// Clear works correctly after popping elements
METHOD ClearAfterPop
VAR
	ReturnedElement : DINT;
END_VAR
IF TestSuite.Test(__POUNAME()).ExecuteTest() THEN
	// Arrange - Push and then pop elements
	fbAnyBuffer.Clear();
	testElement := DINT#100;
	fbAnyBuffer.PushLeft(element := testElement);
	testElement := DINT#200;
	fbAnyBuffer.PushLeft(element := testElement);
	testElement := DINT#200;
	fbAnyBuffer.PushLeft(element := testElement);
	fbAnyBuffer.PopLeft(element := ReturnedElement);
	fbAnyBuffer.PopLeft(element := ReturnedElement);

	// Act
	Success := fbAnyBuffer.Clear();

	// Assert
	TestSuite.Test(__POUNAME()).AssertEqual(TEST_BOOL_TRUE, Success);
	TEST_DINT := 0;
	TestSuite.Test(__POUNAME()).AssertEqual(TEST_DINT, fbAnyBuffer.Metadata.elementCount);
	TestSuite.Test(__POUNAME()).AssertEqual(TEST_DINT, RawBuffer[TEST_LL+0]);
END_IF
END_METHOD

// Clear works correctly after pushing elements
METHOD ClearAfterPush
IF TestSuite.Test(__POUNAME()).ExecuteTest() THEN
	// Arrange - Push some elements first
	fbAnyBuffer.Clear();
	testElement := DINT#100;
	fbAnyBuffer.PushLeft(element := testElement);
	fbAnyBuffer.PushLeft(element := testElement);
	fbAnyBuffer.PushLeft(element := testElement);

	// Act
	Success := fbAnyBuffer.Clear();

	// Assert
	TestSuite.Test(__POUNAME()).AssertEqual(TEST_BOOL_TRUE, Success);
	TEST_DINT := 0;
	TestSuite.Test(__POUNAME()).AssertEqual(TEST_DINT, fbAnyBuffer.Metadata.elementCount);
	TestSuite.Test(__POUNAME()).AssertEqual(TEST_DINT, RawBuffer[TEST_LL+0]);
	TestSuite.Test(__POUNAME()).AssertEqual(TEST_DINT, RawBuffer[TEST_LL+1]);
	TestSuite.Test(__POUNAME()).AssertEqual(TEST_DINT, RawBuffer[TEST_LL+2]);
END_IF
END_METHOD

// Clear on already-empty buffer returns TRUE
METHOD ClearEmptyBuffer
IF TestSuite.Test(__POUNAME()).ExecuteTest() THEN
	// Arrange - Buffer is already empty (elementCount = 0)
	fbAnyBuffer.Clear();

	// Act - Clear again
	Success := fbAnyBuffer.Clear();

	// Assert
	TestSuite.Test(__POUNAME()).AssertEqual(TEST_BOOL_TRUE, Success);
	TEST_DINT := 0;
	TestSuite.Test(__POUNAME()).AssertEqual(TEST_DINT, fbAnyBuffer.Metadata.elementCount);
END_IF
END_METHOD

// Clear works when buffer is at capacity
METHOD ClearFullBuffer
IF TestSuite.Test(__POUNAME()).ExecuteTest() THEN
	// Arrange - Fill buffer to capacity (5 elements)
	RawBuffer[TEST_LL+0] := 100;
	RawBuffer[TEST_LL+1] := 200;
	RawBuffer[TEST_LL+2] := 300;
	RawBuffer[TEST_LL+3] := 400;
	RawBuffer[TEST_LL+4] := 500;
	fbAnyBuffer.Metadata.elementCount := 5;

	// Act
	Success := fbAnyBuffer.Clear();

	// Assert
	TestSuite.Test(__POUNAME()).AssertEqual(TEST_BOOL_TRUE, Success);
	TEST_DINT := 0;
	TestSuite.Test(__POUNAME()).AssertEqual(TEST_DINT, fbAnyBuffer.Metadata.elementCount);
	TestSuite.Test(__POUNAME()).AssertEqual(TEST_DINT, RawBuffer[TEST_LL+0]);
	TestSuite.Test(__POUNAME()).AssertEqual(TEST_DINT, RawBuffer[TEST_LL+1]);
	TestSuite.Test(__POUNAME()).AssertEqual(TEST_DINT, RawBuffer[TEST_LL+2]);
	TestSuite.Test(__POUNAME()).AssertEqual(TEST_DINT, RawBuffer[TEST_LL+3]);
	TestSuite.Test(__POUNAME()).AssertEqual(TEST_DINT, RawBuffer[TEST_LL+4]);
END_IF
END_METHOD

// Clear works when buffer is partially filled
METHOD ClearPartialBuffer
IF TestSuite.Test(__POUNAME()).ExecuteTest() THEN
	// Arrange - Partially fill buffer (2 out of 5 elements)
	RawBuffer[TEST_LL+0] := 100;
	RawBuffer[TEST_LL+1] := 200;
	fbAnyBuffer.Metadata.elementCount := 2;

	// Act
	Success := fbAnyBuffer.Clear();

	// Assert
	TestSuite.Test(__POUNAME()).AssertEqual(TEST_BOOL_TRUE, Success);
	TEST_DINT := 0;
	TestSuite.Test(__POUNAME()).AssertEqual(TEST_DINT, fbAnyBuffer.Metadata.elementCount);
	TestSuite.Test(__POUNAME()).AssertEqual(TEST_DINT, RawBuffer[TEST_LL+0]);
	TestSuite.Test(__POUNAME()).AssertEqual(TEST_DINT, RawBuffer[TEST_LL+1]);
END_IF
END_METHOD

// Clear zeros all buffer positions
METHOD ClearsAllElements
IF TestSuite.Test(__POUNAME()).ExecuteTest() THEN
	// Arrange
	RawBuffer[TEST_LL+0] := 100;
	RawBuffer[TEST_LL+1] := 200;
	RawBuffer[TEST_LL+2] := 300;
	RawBuffer[TEST_LL+3] := 400;
	RawBuffer[TEST_LL+4] := 500;
	fbAnyBuffer.Metadata.elementCount := 5;
	fbAnyBuffer.Metadata.capacity := 0;
	
	// Act
	Success := fbAnyBuffer.Clear();

	// Assert - All buffer positions should be zero
	TEST_DINT := 0;
	TestSuite.Test(__POUNAME()).AssertEqual(TEST_DINT, RawBuffer[TEST_LL+0]);
	TestSuite.Test(__POUNAME()).AssertEqual(TEST_DINT, RawBuffer[TEST_LL+1]);
	TestSuite.Test(__POUNAME()).AssertEqual(TEST_DINT, RawBuffer[TEST_LL+2]);
	TestSuite.Test(__POUNAME()).AssertEqual(TEST_DINT, RawBuffer[TEST_LL+3]);
	TestSuite.Test(__POUNAME()).AssertEqual(TEST_DINT, RawBuffer[TEST_LL+4]);
END_IF
END_METHOD

// Consecutive Clear calls all return TRUE
METHOD MultipleClearCalls
IF TestSuite.Test(__POUNAME()).ExecuteTest() THEN
	// Arrange
	RawBuffer[TEST_LL+0] := 100;
	fbAnyBuffer.Metadata.elementCount := 1;

	// Act - Clear multiple times consecutively
	Success := fbAnyBuffer.Clear();
	TestSuite.Test(__POUNAME()).AssertEqual(TEST_BOOL_TRUE, Success);

	Success := fbAnyBuffer.Clear();
	TestSuite.Test(__POUNAME()).AssertEqual(TEST_BOOL_TRUE, Success);

	Success := fbAnyBuffer.Clear();
	TestSuite.Test(__POUNAME()).AssertEqual(TEST_BOOL_TRUE, Success);

	// Assert - Still returns TRUE and buffer remains clear
	TEST_DINT := 0;
	TestSuite.Test(__POUNAME()).AssertEqual(TEST_DINT, fbAnyBuffer.Metadata.elementCount);
END_IF
END_METHOD

// Clear preserves buffer configuration (capacity, elementSize)
METHOD PreservesConfiguration
VAR
	capacityBefore : DINT;
	elementSizeBefore : DINT;
END_VAR
IF TestSuite.Test(__POUNAME()).ExecuteTest() THEN
	// Arrange
	RawBuffer[TEST_LL+0] := 100;
	fbAnyBuffer.Metadata.elementCount := 1;
	capacityBefore := fbAnyBuffer.Configuration.capacity;
	elementSizeBefore := fbAnyBuffer.Configuration.elementSize;

	// Act
	Success := fbAnyBuffer.Clear();

	// Assert - Configuration should remain unchanged
	TestSuite.Test(__POUNAME()).AssertEqual(capacityBefore, fbAnyBuffer.Configuration.capacity);
	TestSuite.Test(__POUNAME()).AssertEqual(elementSizeBefore, fbAnyBuffer.Configuration.elementSize);
END_IF
END_METHOD

// Clear resets all metadata fields to zero
METHOD ResetsAllMetadata
IF TestSuite.Test(__POUNAME()).ExecuteTest() THEN
	// Arrange
	RawBuffer[TEST_LL+0] := 100;
	RawBuffer[TEST_LL+1] := 200;
	fbAnyBuffer.Metadata.elementCount := 2;
	fbAnyBuffer.Metadata.capacity := 3;

	// Act
	Success := fbAnyBuffer.Clear();

	// Assert - All metadata should be zeroed
	TEST_DINT := 0;
	TestSuite.Test(__POUNAME()).AssertEqual(TEST_DINT, fbAnyBuffer.Metadata.elementCount);
	TEST_DINT := fbAnyBuffer.Configuration.capacity;
	TestSuite.Test(__POUNAME()).AssertEqual(TEST_DINT, fbAnyBuffer.Metadata.capacity);
END_IF
END_METHOD

// Clear resets elementCount to 0
METHOD ResetsElementCount
IF TestSuite.Test(__POUNAME()).ExecuteTest() THEN
	// Arrange
	RawBuffer[TEST_LL+0] := 100;
	RawBuffer[TEST_LL+1] := 200;
	RawBuffer[TEST_LL+2] := 300;
	fbAnyBuffer.Metadata.elementCount := 3;

	// Act
	Success := fbAnyBuffer.Clear();

	// Assert - elementCount should be 0
	TEST_DINT := 0;
	TestSuite.Test(__POUNAME()).AssertEqual(TEST_DINT, fbAnyBuffer.Metadata.elementCount);
END_IF
END_METHOD

// Clear returns TRUE when buffer is initialized
METHOD ReturnsTrue
IF TestSuite.Test(__POUNAME()).ExecuteTest() THEN
	// Arrange
	RawBuffer[TEST_LL+0] := 100;
	fbAnyBuffer.Metadata.elementCount := 1;

	// Act
	Success := fbAnyBuffer.Clear();

	// Assert
	TestSuite.Test(__POUNAME()).AssertEqual(TEST_BOOL_TRUE, Success);
END_IF
END_METHOD

END_PROGRAM

// ---- UnitTests/AnyBuffer/TEST_AnyBuffer_DeleteAtIndex.TcPOU
PROGRAM TEST_AnyBuffer_DeleteAtIndex
VAR
	// Loop counter
	i						: DINT;
END_VAR

DeletesAtValidIndex();
ReturnsTrueOnSuccess();
ReturnsFalseOnInvalidIndex();
RejectsNegativeIndex();
RejectsIndexAtCapacity();
RejectsIndexAboveCapacity();
ExtremeBounds();
DeleteAtZero();
DeleteAtCapacityMinusOne();
DeleteAllPositions();
PreservesOtherData();
DeleteAlreadyEmpty();
DeleteDoesNotShift();
DeleteWhenEmpty();
MetadataUnchanged();
ConsecutiveDeletesSamePosition();

// Multiple deletes at same position succeed without metadata changes
METHOD ConsecutiveDeletesSamePosition
IF TestSuite.Test(__POUNAME()).ExecuteTest() THEN
	// Arrange
	fbAnyBuffer.Clear();
	RawBuffer[TEST_LL+2] := 9999;
	fbAnyBuffer.Metadata.elementCount := 5;

	// Act & Assert - first delete
	Success := fbAnyBuffer.DeleteAtIndex(index := TEST_LL+2);
	TestSuite.Test(__POUNAME()).AssertEqual(TEST_BOOL_TRUE, Success);
	TEST_DINT := 0;
	TestSuite.Test(__POUNAME()).AssertEqual(TEST_DINT, RawBuffer[TEST_LL+2]);
	// Metadata should remain unchanged
	TEST_DINT := 5;
	TestSuite.Test(__POUNAME()).AssertEqual(TEST_DINT, fbAnyBuffer.Metadata.elementCount);

	// Act & Assert - second delete at same position (already zero)
	RawBuffer[TEST_LL+2] := 8888;  // Set to non-zero to test clearing
	Success := fbAnyBuffer.DeleteAtIndex(index := TEST_LL+2);
	TestSuite.Test(__POUNAME()).AssertEqual(TEST_BOOL_TRUE, Success);
	TEST_DINT := 0;
	TestSuite.Test(__POUNAME()).AssertEqual(TEST_DINT, RawBuffer[TEST_LL+2]);
	// Metadata should remain unchanged
	TEST_DINT := 5;
	TestSuite.Test(__POUNAME()).AssertEqual(TEST_DINT, fbAnyBuffer.Metadata.elementCount);

	// Act & Assert - third delete at same position
	RawBuffer[TEST_LL+2] := 7777;  // Set to non-zero again
	Success := fbAnyBuffer.DeleteAtIndex(index := TEST_LL+2);
	TestSuite.Test(__POUNAME()).AssertEqual(TEST_BOOL_TRUE, Success);
	TEST_DINT := 0;
	TestSuite.Test(__POUNAME()).AssertEqual(TEST_DINT, RawBuffer[TEST_LL+2]);
	// Metadata should STILL remain unchanged
	TEST_DINT := 5;
	TestSuite.Test(__POUNAME()).AssertEqual(TEST_DINT, fbAnyBuffer.Metadata.elementCount);
END_IF
END_METHOD

// DeleteAtIndex works correctly at all valid indices (0 through capacity-1)
METHOD DeleteAllPositions
IF TestSuite.Test(__POUNAME()).ExecuteTest() THEN
	// Arrange - fill all positions with distinct values
	fbAnyBuffer.Clear();
	FOR i := TEST_LL TO TEST_UL DO
		RawBuffer[i] := (i - TEST_LL + 1) * 1000;  // 1000, 2000, 3000, 4000, 5000
	END_FOR
	fbAnyBuffer.Metadata.elementCount := 5;

	// Act & Assert - delete each position and verify it's cleared
	FOR i := TEST_LL TO TEST_UL DO
		Success := fbAnyBuffer.DeleteAtIndex(index := i);
		TestSuite.Test(__POUNAME()).AssertEqual(TEST_BOOL_TRUE, Success);
		TEST_DINT := 0;
		TestSuite.Test(__POUNAME()).AssertEqual(TEST_DINT, RawBuffer[i]);
	END_FOR
END_IF
END_METHOD

// Deleting an already-cleared position returns TRUE and remains zero
METHOD DeleteAlreadyEmpty
IF TestSuite.Test(__POUNAME()).ExecuteTest() THEN
	// Arrange - clear buffer so all positions are zero
	fbAnyBuffer.Clear();

	// Verify position is already zero
	TEST_DINT := 0;
	TestSuite.Test(__POUNAME()).AssertEqual(TEST_DINT, RawBuffer[TEST_LL+2]);

	// Act - delete at already empty position
	Success := fbAnyBuffer.DeleteAtIndex(index := TEST_LL+2);

	// Assert - should return TRUE
	TestSuite.Test(__POUNAME()).AssertEqual(TEST_BOOL_TRUE, Success);

	// Assert - position should still be zero
	TEST_DINT := 0;
	TestSuite.Test(__POUNAME()).AssertEqual(TEST_DINT, RawBuffer[TEST_LL+2]);
END_IF
END_METHOD

// DeleteAtIndex at last position (capacity-1) works correctly
METHOD DeleteAtCapacityMinusOne
IF TestSuite.Test(__POUNAME()).ExecuteTest() THEN
	// Arrange - capacity is 5, last valid index is 4
	fbAnyBuffer.Clear();
	RawBuffer[TEST_LL+4] := 5000;
	fbAnyBuffer.Metadata.elementCount := 1;

	// Act
	Success := fbAnyBuffer.DeleteAtIndex(index := TEST_LL+4);

	// Assert - position cleared, metadata unchanged
	TestSuite.Test(__POUNAME()).AssertEqual(TEST_BOOL_TRUE, Success);
	TEST_DINT := 0;
	TestSuite.Test(__POUNAME()).AssertEqual(TEST_DINT, RawBuffer[TEST_LL+4]);
	// Metadata should remain unchanged
	TEST_DINT := 1;
	TestSuite.Test(__POUNAME()).AssertEqual(TEST_DINT, fbAnyBuffer.Metadata.elementCount);
END_IF
END_METHOD

// DeleteAtIndex at first position (index 0) works correctly
METHOD DeleteAtZero
IF TestSuite.Test(__POUNAME()).ExecuteTest() THEN
	// Arrange
	fbAnyBuffer.Clear();
	RawBuffer[TEST_LL] := 1000;
	fbAnyBuffer.Metadata.elementCount := 1;

	// Act
	Success := fbAnyBuffer.DeleteAtIndex(index := TEST_LL);

	// Assert - position cleared, metadata unchanged
	TestSuite.Test(__POUNAME()).AssertEqual(TEST_BOOL_TRUE, Success);
	TEST_DINT := 0;
	TestSuite.Test(__POUNAME()).AssertEqual(TEST_DINT, RawBuffer[TEST_LL]);
	// Metadata should remain unchanged
	TEST_DINT := 1;
	TestSuite.Test(__POUNAME()).AssertEqual(TEST_DINT, fbAnyBuffer.Metadata.elementCount);
END_IF
END_METHOD

// Elements after deleted index remain at their original positions
METHOD DeleteDoesNotShift
IF TestSuite.Test(__POUNAME()).ExecuteTest() THEN
	// Arrange - fill all positions with distinct values
	fbAnyBuffer.Clear();
	RawBuffer[TEST_LL+0] := 100;
	RawBuffer[TEST_LL+1] := 200;
	RawBuffer[TEST_LL+2] := 300;
	RawBuffer[TEST_LL+3] := 400;
	RawBuffer[TEST_LL+4] := 500;
	fbAnyBuffer.Metadata.elementCount := 5;

	// Act - delete at index 1
	Success := fbAnyBuffer.DeleteAtIndex(index := TEST_LL+1);

	// Assert - deleted position is zero
	TEST_DINT := 0;
	TestSuite.Test(__POUNAME()).AssertEqual(TEST_DINT, RawBuffer[TEST_LL+1]);

	// Assert - elements after deleted index remain at their original positions (NO SHIFT)
	TEST_DINT := 100;
	TestSuite.Test(__POUNAME()).AssertEqual(TEST_DINT, RawBuffer[TEST_LL+0]);
	TEST_DINT := 300;
	TestSuite.Test(__POUNAME()).AssertEqual(TEST_DINT, RawBuffer[TEST_LL+2]);  // Still at position 2
	TEST_DINT := 400;
	TestSuite.Test(__POUNAME()).AssertEqual(TEST_DINT, RawBuffer[TEST_LL+3]);  // Still at position 3
	TEST_DINT := 500;
	TestSuite.Test(__POUNAME()).AssertEqual(TEST_DINT, RawBuffer[TEST_LL+4]);  // Still at position 4
END_IF
END_METHOD

// DeleteAtIndex zeros element at valid index
METHOD DeletesAtValidIndex
IF TestSuite.Test(__POUNAME()).ExecuteTest() THEN
	// Arrange
	fbAnyBuffer.Clear();
	RawBuffer[TEST_LL+2] := 9999;
	fbAnyBuffer.Metadata.elementCount := 1;

	// Act
	Success := fbAnyBuffer.DeleteAtIndex(index := TEST_LL+2);

	// Assert
	TestSuite.Test(__POUNAME()).AssertEqual(TEST_BOOL_TRUE, Success);
	TEST_DINT := 0;
	TestSuite.Test(__POUNAME()).AssertEqual(TEST_DINT, RawBuffer[TEST_LL+2]);
END_IF
END_METHOD

// Deletion succeeds even when elementCount is 0 (clears position only)
METHOD DeleteWhenEmpty
IF TestSuite.Test(__POUNAME()).ExecuteTest() THEN
	// Arrange - clear buffer (elementCount = 0)
	fbAnyBuffer.Clear();
	RawBuffer[TEST_LL+2] := 9999;  // Manually set a position to non-zero
	fbAnyBuffer.Metadata.elementCount := 0;

	// Act - delete when elementCount is 0
	Success := fbAnyBuffer.DeleteAtIndex(index := TEST_LL+2);

	// Assert - should succeed (clears position)
	TestSuite.Test(__POUNAME()).AssertEqual(TEST_BOOL_TRUE, Success);
	TEST_DINT := 0;
	TestSuite.Test(__POUNAME()).AssertEqual(TEST_DINT, RawBuffer[TEST_LL+2]);

	// Note: elementCount will decrement to -1, which may need handling
	// This test documents current behavior
END_IF
END_METHOD

// DeleteAtIndex rejects extreme index values
METHOD ExtremeBounds
IF TestSuite.Test(__POUNAME()).ExecuteTest() THEN
	// Act & Assert - very large negative index
	Success := fbAnyBuffer.DeleteAtIndex(index := -10000);
	TestSuite.Test(__POUNAME()).AssertEqual(TEST_BOOL_FALSE, Success);

	// Act & Assert - very large positive index
	Success := fbAnyBuffer.DeleteAtIndex(index := 10000);
	TestSuite.Test(__POUNAME()).AssertEqual(TEST_BOOL_FALSE, Success);

	// Act & Assert - maximum DINT value
	Success := fbAnyBuffer.DeleteAtIndex(index := 16#7FFFFFFF);
	TestSuite.Test(__POUNAME()).AssertEqual(TEST_BOOL_FALSE, Success);

	// Act & Assert - minimum DINT value
	Success := fbAnyBuffer.DeleteAtIndex(index := -16#7FFFFFFF);
	TestSuite.Test(__POUNAME()).AssertEqual(TEST_BOOL_FALSE, Success);
END_IF
END_METHOD

// ElementCount and all metadata remain unchanged after deletion
METHOD MetadataUnchanged
IF TestSuite.Test(__POUNAME()).ExecuteTest() THEN
	// Arrange
	fbAnyBuffer.Clear();
	RawBuffer[TEST_LL+0] := 100;
	RawBuffer[TEST_LL+1] := 200;
	RawBuffer[TEST_LL+2] := 300;
	RawBuffer[TEST_LL+3] := 400;
	RawBuffer[TEST_LL+4] := 500;
	fbAnyBuffer.Metadata.elementCount := 5;
	fbAnyBuffer.Metadata.capacity := 0;  // Set to 0 for this test

	// Act - delete at various indices
	Success := fbAnyBuffer.DeleteAtIndex(index := TEST_LL+1);
	TestSuite.Test(__POUNAME()).AssertEqual(TEST_BOOL_TRUE, Success);
	TEST_DINT := 0;
	TestSuite.Test(__POUNAME()).AssertEqual(TEST_DINT, RawBuffer[TEST_LL+1]);

	// Assert - metadata should remain completely unchanged
	TEST_DINT := 5;
	TestSuite.Test(__POUNAME()).AssertEqual(TEST_DINT, fbAnyBuffer.Metadata.elementCount);
	TEST_DINT := 0;
	TestSuite.Test(__POUNAME()).AssertEqual(TEST_DINT, fbAnyBuffer.Metadata.capacity);

	// Act - delete another position
	Success := fbAnyBuffer.DeleteAtIndex(index := TEST_LL+3);
	TestSuite.Test(__POUNAME()).AssertEqual(TEST_BOOL_TRUE, Success);
	TEST_DINT := 0;
	TestSuite.Test(__POUNAME()).AssertEqual(TEST_DINT, RawBuffer[TEST_LL+3]);

	// Assert - metadata should STILL be unchanged
	TEST_DINT := 5;
	TestSuite.Test(__POUNAME()).AssertEqual(TEST_DINT, fbAnyBuffer.Metadata.elementCount);
	TEST_DINT := 0;
	TestSuite.Test(__POUNAME()).AssertEqual(TEST_DINT, fbAnyBuffer.Metadata.capacity);
END_IF
END_METHOD

// Deletion at one index does not affect data at other indices
METHOD PreservesOtherData
IF TestSuite.Test(__POUNAME()).ExecuteTest() THEN
	// Arrange - fill all positions with distinct values
	fbAnyBuffer.Clear();
	RawBuffer[TEST_LL+0] := 1000;
	RawBuffer[TEST_LL+1] := 2000;
	RawBuffer[TEST_LL+2] := 3000;
	RawBuffer[TEST_LL+3] := 4000;
	RawBuffer[TEST_LL+4] := 5000;
	fbAnyBuffer.Metadata.elementCount := 5;

	// Act - delete middle position
	Success := fbAnyBuffer.DeleteAtIndex(index := TEST_LL+2);
	TestSuite.Test(__POUNAME()).AssertEqual(TEST_BOOL_TRUE, Success);

	// Assert - deleted position is cleared
	TEST_DINT := 0;
	TestSuite.Test(__POUNAME()).AssertEqual(TEST_DINT, RawBuffer[TEST_LL+2]);

	// Assert - other positions are preserved
	TEST_DINT := 1000;
	TestSuite.Test(__POUNAME()).AssertEqual(TEST_DINT, RawBuffer[TEST_LL+0]);
	TEST_DINT := 2000;
	TestSuite.Test(__POUNAME()).AssertEqual(TEST_DINT, RawBuffer[TEST_LL+1]);
	TEST_DINT := 4000;
	TestSuite.Test(__POUNAME()).AssertEqual(TEST_DINT, RawBuffer[TEST_LL+3]);
	TEST_DINT := 5000;
	TestSuite.Test(__POUNAME()).AssertEqual(TEST_DINT, RawBuffer[TEST_LL+4]);
END_IF
END_METHOD

// DeleteAtIndex rejects index > capacity with error log
METHOD RejectsIndexAboveCapacity
IF TestSuite.Test(__POUNAME()).ExecuteTest() THEN
	// Arrange - capacity is 5

	// Act - try to delete at index 10 (above capacity)
	Success := fbAnyBuffer.DeleteAtIndex(index := TEST_UL+10);

	// Assert
	TestSuite.Test(__POUNAME()).AssertEqual(TEST_BOOL_FALSE, Success);
END_IF
END_METHOD

// DeleteAtIndex rejects index == capacity with error log
METHOD RejectsIndexAtCapacity
IF TestSuite.Test(__POUNAME()).ExecuteTest() THEN
	// Arrange - capacity is TEST_UL-TEST_LL+1 

	// Act - try to delete at index TEST_UL (equals capacity)
	Success := fbAnyBuffer.DeleteAtIndex(index := TEST_UL+1);

	// Assert
	TestSuite.Test(__POUNAME()).AssertEqual(TEST_BOOL_FALSE, Success);
END_IF
END_METHOD

// DeleteAtIndex rejects index < 0 with error log
METHOD RejectsNegativeIndex
IF TestSuite.Test(__POUNAME()).ExecuteTest() THEN
	// Act
	Success := fbAnyBuffer.DeleteAtIndex(index := TEST_LL+-1);

	// Assert
	TestSuite.Test(__POUNAME()).AssertEqual(TEST_BOOL_FALSE, Success);
END_IF
END_METHOD

// DeleteAtIndex returns FALSE for out-of-bounds index
METHOD ReturnsFalseOnInvalidIndex
IF TestSuite.Test(__POUNAME()).ExecuteTest() THEN
	// Act & Assert - negative index
	Success := fbAnyBuffer.DeleteAtIndex(index := TEST_LL-1);
	TestSuite.Test(__POUNAME()).AssertEqual(TEST_BOOL_FALSE, Success);

	// Act & Assert - index at capacity
	Success := fbAnyBuffer.DeleteAtIndex(index := TEST_UL+1);
	TestSuite.Test(__POUNAME()).AssertEqual(TEST_BOOL_FALSE, Success);

	// Act & Assert - index above capacity
	Success := fbAnyBuffer.DeleteAtIndex(index := TEST_UL+100);
	TestSuite.Test(__POUNAME()).AssertEqual(TEST_BOOL_FALSE, Success);
END_IF
END_METHOD

// DeleteAtIndex returns TRUE when deletion succeeds
METHOD ReturnsTrueOnSuccess
IF TestSuite.Test(__POUNAME()).ExecuteTest() THEN
	// Arrange
	fbAnyBuffer.Clear();
	RawBuffer[TEST_LL] := 100;
	fbAnyBuffer.Metadata.elementCount := 1;

	// Act
	Success := fbAnyBuffer.DeleteAtIndex(index := TEST_LL);

	// Assert
	TestSuite.Test(__POUNAME()).AssertEqual(TEST_BOOL_TRUE, Success);
END_IF
END_METHOD

END_PROGRAM

// ---- UnitTests/AnyBuffer/TEST_AnyBuffer_InsertAtIndex.TcPOU
PROGRAM TEST_AnyBuffer_InsertAtIndex
VAR
	// Loop counter
	i						: DINT;
END_VAR

InsertAtBeginning();
InsertInMiddle();
InsertAtEnd();
InsertIntoEmptyBuffer();
ReturnsTrueOnSuccess();
ReturnsFalseOnNegativeIndex();
ReturnsFalseOnIndexOutOfBounds();
ReturnsFalseOnFullBuffer();
WrongElementSize();
IncrementsElementCount();
ShiftsElementsCorrectly();
PreservesElementOrder();
MultipleInsertions();
InsertAllValidPositions();
InsertAtIndexEquivalentToAppendLeft();
InsertAtIndexEquivalentToAppendRight();

// Element count increases by 1 after insert
METHOD IncrementsElementCount
IF TestSuite.Test(__POUNAME()).ExecuteTest() THEN
	// Arrange
	fbAnyBuffer.Clear();
	testElement := DINT#100;
	fbAnyBuffer.PushRight(element := testElement);
	testElement := DINT#200;
	fbAnyBuffer.PushRight(element := testElement);
	TEST_DINT := 2;
	TestSuite.Test(__POUNAME()).AssertEqual(TEST_DINT, fbAnyBuffer.Metadata.elementCount);

	// Act - Insert at middle
	testElement := DINT#150;
	Success := fbAnyBuffer.PushAtIndex(index := TEST_LL+1, element := testElement);

	// Assert
	TestSuite.Test(__POUNAME()).AssertEqual(TEST_BOOL_TRUE, Success);
	TEST_DINT := 3;
	TestSuite.Test(__POUNAME()).AssertEqual(TEST_DINT, fbAnyBuffer.Metadata.elementCount);
END_IF
END_METHOD

// Can insert at every valid position (0 to elementCount)
METHOD InsertAllValidPositions
IF TestSuite.Test(__POUNAME()).ExecuteTest() THEN
	// Arrange - Start with one element
	fbAnyBuffer.Clear();
	testElement := DINT#1000;
	fbAnyBuffer.PushRight(element := testElement);

	// Act & Assert - Insert at position 0 (before existing element)
	testElement := DINT#500;
	Success := fbAnyBuffer.PushAtIndex(index := TEST_LL, element := testElement);
	TestSuite.Test(__POUNAME()).AssertEqual(TEST_BOOL_TRUE, Success);
	TEST_DINT := 2;
	TestSuite.Test(__POUNAME()).AssertEqual(TEST_DINT, fbAnyBuffer.Metadata.elementCount);

	// Insert at position 1 (middle)
	testElement := DINT#750;
	Success := fbAnyBuffer.PushAtIndex(index := TEST_LL+1, element := testElement);
	TestSuite.Test(__POUNAME()).AssertEqual(TEST_BOOL_TRUE, Success);
	TEST_DINT := 3;
	TestSuite.Test(__POUNAME()).AssertEqual(TEST_DINT, fbAnyBuffer.Metadata.elementCount);

	// Insert at position 3 (end)
	testElement := DINT#1500;
	Success := fbAnyBuffer.PushAtIndex(index := TEST_LL+3, element := testElement);
	TestSuite.Test(__POUNAME()).AssertEqual(TEST_BOOL_TRUE, Success);
	TEST_DINT := 4;
	TestSuite.Test(__POUNAME()).AssertEqual(TEST_DINT, fbAnyBuffer.Metadata.elementCount);

	// Verify final order: [500, 750, 1000, 1500]
	TEST_DINT := 500;
	TestSuite.Test(__POUNAME()).AssertEqual(TEST_DINT, RawBuffer[TEST_LL+0]);
	TEST_DINT := 750;
	TestSuite.Test(__POUNAME()).AssertEqual(TEST_DINT, RawBuffer[TEST_LL+1]);
	TEST_DINT := 1000;
	TestSuite.Test(__POUNAME()).AssertEqual(TEST_DINT, RawBuffer[TEST_LL+2]);
	TEST_DINT := 1500;
	TestSuite.Test(__POUNAME()).AssertEqual(TEST_DINT, RawBuffer[TEST_LL+3]);
END_IF
END_METHOD

// Inserting at index 0 shifts all elements and inserts at front
METHOD InsertAtBeginning
IF TestSuite.Test(__POUNAME()).ExecuteTest() THEN
	// Arrange - [100, 200, 300]
	fbAnyBuffer.Clear();
	testElement := DINT#100;
	fbAnyBuffer.PushRight(element := testElement);
	testElement := DINT#200;
	fbAnyBuffer.PushRight(element := testElement);
	testElement := DINT#300;
	fbAnyBuffer.PushRight(element := testElement);

	// Act - Insert 50 at beginning
	testElement := DINT#50;
	Success := fbAnyBuffer.PushAtIndex(index := TEST_LL, element := testElement);

	// Assert - [50, 100, 200, 300]
	TestSuite.Test(__POUNAME()).AssertEqual(TEST_BOOL_TRUE, Success);
	TEST_DINT := 50;
	TestSuite.Test(__POUNAME()).AssertEqual(TEST_DINT, RawBuffer[TEST_LL+0]);
	TEST_DINT := 100;
	TestSuite.Test(__POUNAME()).AssertEqual(TEST_DINT, RawBuffer[TEST_LL+1]);
	TEST_DINT := 200;
	TestSuite.Test(__POUNAME()).AssertEqual(TEST_DINT, RawBuffer[TEST_LL+2]);
	TEST_DINT := 300;
	TestSuite.Test(__POUNAME()).AssertEqual(TEST_DINT, RawBuffer[TEST_LL+3]);
	TEST_DINT := 4;
	TestSuite.Test(__POUNAME()).AssertEqual(TEST_DINT, fbAnyBuffer.Metadata.elementCount);
END_IF
END_METHOD

// Inserting at index elementCount appends at end (like AppendRight)
METHOD InsertAtEnd
IF TestSuite.Test(__POUNAME()).ExecuteTest() THEN
	// Arrange - [100, 200, 300]
	fbAnyBuffer.Clear();
	testElement := DINT#100;
	fbAnyBuffer.PushRight(element := testElement);
	testElement := DINT#200;
	fbAnyBuffer.PushRight(element := testElement);
	testElement := DINT#300;
	fbAnyBuffer.PushRight(element := testElement);

	// Act - Insert 400 at end (index 3 = elementCount)
	testElement := DINT#400;
	Success := fbAnyBuffer.PushAtIndex(index := TEST_LL+3, element := testElement);

	// Assert - [100, 200, 300, 400]
	TestSuite.Test(__POUNAME()).AssertEqual(TEST_BOOL_TRUE, Success);
	TEST_DINT := 100;
	TestSuite.Test(__POUNAME()).AssertEqual(TEST_DINT, RawBuffer[TEST_LL+0]);
	TEST_DINT := 200;
	TestSuite.Test(__POUNAME()).AssertEqual(TEST_DINT, RawBuffer[TEST_LL+1]);
	TEST_DINT := 300;
	TestSuite.Test(__POUNAME()).AssertEqual(TEST_DINT, RawBuffer[TEST_LL+2]);
	TEST_DINT := 400;
	TestSuite.Test(__POUNAME()).AssertEqual(TEST_DINT, RawBuffer[TEST_LL+3]);
	TEST_DINT := 4;
	TestSuite.Test(__POUNAME()).AssertEqual(TEST_DINT, fbAnyBuffer.Metadata.elementCount);
END_IF
END_METHOD

// InsertAtIndex(0) behaves same as AppendLeft
METHOD InsertAtIndexEquivalentToAppendLeft
IF TestSuite.Test(__POUNAME()).ExecuteTest() THEN
	// Arrange - Two buffers with same initial state
	fbAnyBuffer.Clear();
	testElement := DINT#100;
	fbAnyBuffer.PushRight(element := testElement);
	testElement := DINT#200;
	fbAnyBuffer.PushRight(element := testElement);

	// Use a second buffer for comparison
	fbCompareBuffer.Clear();
	testElement := DINT#100;
	fbCompareBuffer.PushRight(element := testElement);
	testElement := DINT#200;
	fbCompareBuffer.PushRight(element := testElement);

	// Act - InsertAtIndex(0) vs AppendLeft
	testElement := DINT#50;
	Success := fbAnyBuffer.PushAtIndex(index := TEST_LL, element := testElement);
	TestSuite.Test(__POUNAME()).AssertEqual(TEST_BOOL_TRUE, Success);

	testElement := DINT#50;
	fbCompareBuffer.PushLeft(element := testElement);

	// Assert - Both buffers should be identical
	TEST_DINT := 3;
	TestSuite.Test(__POUNAME()).AssertEqual(TEST_DINT, fbAnyBuffer.Metadata.elementCount);
	TestSuite.Test(__POUNAME()).AssertEqual(TEST_DINT, fbCompareBuffer.Metadata.elementCount);

	TEST_DINT := 50;
	TestSuite.Test(__POUNAME()).AssertEqual(TEST_DINT, RawBuffer[TEST_LL+0]);
	TestSuite.Test(__POUNAME()).AssertEqual(TEST_DINT, CompareBuffer[TEST_LL+0]);

	TEST_DINT := 100;
	TestSuite.Test(__POUNAME()).AssertEqual(TEST_DINT, RawBuffer[TEST_LL+1]);
	TestSuite.Test(__POUNAME()).AssertEqual(TEST_DINT, CompareBuffer[TEST_LL+1]);

	TEST_DINT := 200;
	TestSuite.Test(__POUNAME()).AssertEqual(TEST_DINT, RawBuffer[TEST_LL+2]);
	TestSuite.Test(__POUNAME()).AssertEqual(TEST_DINT, CompareBuffer[TEST_LL+2]);
END_IF
END_METHOD

// InsertAtIndex(elementCount) behaves same as AppendRight
METHOD InsertAtIndexEquivalentToAppendRight
IF TestSuite.Test(__POUNAME()).ExecuteTest() THEN
	// Arrange - Two buffers with same initial state
	fbAnyBuffer.Clear();
	testElement := DINT#100;
	fbAnyBuffer.PushRight(element := testElement);
	testElement := DINT#200;
	fbAnyBuffer.PushRight(element := testElement);

	// Use a second buffer for comparison
	fbCompareBuffer.Clear();
	testElement := DINT#100;
	fbCompareBuffer.PushRight(element := testElement);
	testElement := DINT#200;
	fbCompareBuffer.PushRight(element := testElement);

	// Act - InsertAtIndex(elementCount) vs AppendRight
	testElement := DINT#300;
	Success := fbAnyBuffer.PushAtIndex(index := TEST_LL+2, element := testElement);  // elementCount = 2
	TestSuite.Test(__POUNAME()).AssertEqual(TEST_BOOL_TRUE, Success);

	testElement := DINT#300;
	fbCompareBuffer.PushRight(element := testElement);

	// Assert - Both buffers should be identical
	TEST_DINT := 3;
	TestSuite.Test(__POUNAME()).AssertEqual(TEST_DINT, fbAnyBuffer.Metadata.elementCount);
	TestSuite.Test(__POUNAME()).AssertEqual(TEST_DINT, fbCompareBuffer.Metadata.elementCount);

	TEST_DINT := 100;
	TestSuite.Test(__POUNAME()).AssertEqual(TEST_DINT, RawBuffer[TEST_LL+0]);
	TestSuite.Test(__POUNAME()).AssertEqual(TEST_DINT, CompareBuffer[TEST_LL+0]);

	TEST_DINT := 200;
	TestSuite.Test(__POUNAME()).AssertEqual(TEST_DINT, RawBuffer[TEST_LL+1]);
	TestSuite.Test(__POUNAME()).AssertEqual(TEST_DINT, CompareBuffer[TEST_LL+1]);

	TEST_DINT := 300;
	TestSuite.Test(__POUNAME()).AssertEqual(TEST_DINT, RawBuffer[TEST_LL+2]);
	TestSuite.Test(__POUNAME()).AssertEqual(TEST_DINT, CompareBuffer[TEST_LL+2]);
END_IF
END_METHOD

// Inserting at middle index shifts remaining elements correctly
METHOD InsertInMiddle
IF TestSuite.Test(__POUNAME()).ExecuteTest() THEN
	// Arrange - [100, 300]
	fbAnyBuffer.Clear();
	testElement := DINT#100;
	fbAnyBuffer.PushRight(element := testElement);
	testElement := DINT#300;
	fbAnyBuffer.PushRight(element := testElement);

	// Act - Insert 200 in middle (index 1)
	testElement := DINT#200;
	Success := fbAnyBuffer.PushAtIndex(index := TEST_LL+1, element := testElement);

	// Assert - [100, 200, 300]
	TestSuite.Test(__POUNAME()).AssertEqual(TEST_BOOL_TRUE, Success);
	TEST_DINT := 100;
	TestSuite.Test(__POUNAME()).AssertEqual(TEST_DINT, RawBuffer[TEST_LL+0]);
	TEST_DINT := 200;
	TestSuite.Test(__POUNAME()).AssertEqual(TEST_DINT, RawBuffer[TEST_LL+1]);
	TEST_DINT := 300;
	TestSuite.Test(__POUNAME()).AssertEqual(TEST_DINT, RawBuffer[TEST_LL+2]);
	TEST_DINT := 3;
	TestSuite.Test(__POUNAME()).AssertEqual(TEST_DINT, fbAnyBuffer.Metadata.elementCount);
END_IF
END_METHOD

// Inserting at index 0 in empty buffer works
METHOD InsertIntoEmptyBuffer
IF TestSuite.Test(__POUNAME()).ExecuteTest() THEN
	// Arrange
	fbAnyBuffer.Clear();

	// Act - Insert into empty buffer
	testElement := DINT#100;
	Success := fbAnyBuffer.PushAtIndex(index := TEST_LL, element := testElement);

	// Assert - [100]
	TestSuite.Test(__POUNAME()).AssertEqual(TEST_BOOL_TRUE, Success);
	TEST_DINT := 100;
	TestSuite.Test(__POUNAME()).AssertEqual(TEST_DINT, RawBuffer[TEST_LL]);
	TEST_DINT := 1;
	TestSuite.Test(__POUNAME()).AssertEqual(TEST_DINT, fbAnyBuffer.Metadata.elementCount);
END_IF
END_METHOD

// Sequential insertions at different indices work correctly
METHOD MultipleInsertions
IF TestSuite.Test(__POUNAME()).ExecuteTest() THEN
	// Arrange
	fbAnyBuffer.Clear();
	testElement := DINT#100;
	fbAnyBuffer.PushRight(element := testElement);
	testElement := DINT#400;
	fbAnyBuffer.PushRight(element := testElement);

	// Act - Multiple inserts
	testElement := DINT#200;
	Success := fbAnyBuffer.PushAtIndex(index := TEST_LL+1, element := testElement);
	TestSuite.Test(__POUNAME()).AssertEqual(TEST_BOOL_TRUE, Success);

	testElement := DINT#300;
	Success := fbAnyBuffer.PushAtIndex(index := TEST_LL+2, element := testElement);
	TestSuite.Test(__POUNAME()).AssertEqual(TEST_BOOL_TRUE, Success);

	testElement := DINT#500;
	Success := fbAnyBuffer.PushAtIndex(index := TEST_LL+4, element := testElement);
	TestSuite.Test(__POUNAME()).AssertEqual(TEST_BOOL_TRUE, Success);

	// Assert - [100, 200, 300, 400, 500]
	TEST_DINT := 5;
	TestSuite.Test(__POUNAME()).AssertEqual(TEST_DINT, fbAnyBuffer.Metadata.elementCount);
	TEST_DINT := 100;
	TestSuite.Test(__POUNAME()).AssertEqual(TEST_DINT, RawBuffer[TEST_LL+0]);
	TEST_DINT := 200;
	TestSuite.Test(__POUNAME()).AssertEqual(TEST_DINT, RawBuffer[TEST_LL+1]);
	TEST_DINT := 300;
	TestSuite.Test(__POUNAME()).AssertEqual(TEST_DINT, RawBuffer[TEST_LL+2]);
	TEST_DINT := 400;
	TestSuite.Test(__POUNAME()).AssertEqual(TEST_DINT, RawBuffer[TEST_LL+3]);
	TEST_DINT := 500;
	TestSuite.Test(__POUNAME()).AssertEqual(TEST_DINT, RawBuffer[TEST_LL+4]);
END_IF
END_METHOD

// Element order is preserved after insert
METHOD PreservesElementOrder
IF TestSuite.Test(__POUNAME()).ExecuteTest() THEN
	// Arrange - [10, 20, 30, 40, 50]
	fbAnyBuffer.Clear();
	FOR i := 1 TO 5 DO
		testElement := TO_DINT(i * 10);
		fbAnyBuffer.PushRight(element := testElement);
	END_FOR

	// Act - Insert 25 between 20 and 30 (index 2)
	testElement := DINT#25;
	Success := fbAnyBuffer.PushAtIndex(index := TEST_LL+2, element := testElement);

	// Assert - [10, 20, 25, 30, 40] (50 dropped due to capacity)
	// Wait, buffer has capacity 5, so after 5 elements it's full
	// Actually with capacity 5 (0..4), we can't add a 6th element
	// Let me reconsider: start with 4 elements, then insert
	fbAnyBuffer.Clear();
	testElement := DINT#10;
	fbAnyBuffer.PushRight(element := testElement);
	testElement := DINT#20;
	fbAnyBuffer.PushRight(element := testElement);
	testElement := DINT#30;
	fbAnyBuffer.PushRight(element := testElement);
	testElement := DINT#40;
	fbAnyBuffer.PushRight(element := testElement);

	// Insert 25 between 20 and 30
	testElement := DINT#25;
	Success := fbAnyBuffer.PushAtIndex(index := TEST_LL+2, element := testElement);

	// Assert - [10, 20, 25, 30, 40]
	TestSuite.Test(__POUNAME()).AssertEqual(TEST_BOOL_TRUE, Success);
	TEST_DINT := 5;
	TestSuite.Test(__POUNAME()).AssertEqual(TEST_DINT, fbAnyBuffer.Metadata.elementCount);
	TEST_DINT := 10;
	TestSuite.Test(__POUNAME()).AssertEqual(TEST_DINT, RawBuffer[TEST_LL+0]);
	TEST_DINT := 20;
	TestSuite.Test(__POUNAME()).AssertEqual(TEST_DINT, RawBuffer[TEST_LL+1]);
	TEST_DINT := 25;
	TestSuite.Test(__POUNAME()).AssertEqual(TEST_DINT, RawBuffer[TEST_LL+2]);
	TEST_DINT := 30;
	TestSuite.Test(__POUNAME()).AssertEqual(TEST_DINT, RawBuffer[TEST_LL+3]);
	TEST_DINT := 40;
	TestSuite.Test(__POUNAME()).AssertEqual(TEST_DINT, RawBuffer[TEST_LL+4]);
END_IF
END_METHOD

// FALSE returned when buffer is at capacity
METHOD ReturnsFalseOnFullBuffer
IF TestSuite.Test(__POUNAME()).ExecuteTest() THEN
	// Arrange - Fill buffer to capacity
	fbAnyBuffer.Clear();
	FOR i := 1 TO 5 DO
		testElement := TO_DINT(i * 100);
		fbAnyBuffer.PushRight(element := testElement);
	END_FOR
	TEST_DINT := 5;
	TestSuite.Test(__POUNAME()).AssertEqual(TEST_DINT, fbAnyBuffer.Metadata.elementCount);

	// Act - Try to insert into full buffer
	testElement := DINT#999;
	Success := fbAnyBuffer.PushAtIndex(index := TEST_LL+2, element := testElement);

	// Assert
	TestSuite.Test(__POUNAME()).AssertEqual(TEST_BOOL_FALSE, Success);
	TEST_DINT := 5;
	TestSuite.Test(__POUNAME()).AssertEqual(TEST_DINT, fbAnyBuffer.Metadata.elementCount);
END_IF
END_METHOD

// FALSE returned when index > elementCount
METHOD ReturnsFalseOnIndexOutOfBounds
IF TestSuite.Test(__POUNAME()).ExecuteTest() THEN
	// Arrange
	fbAnyBuffer.Clear();
	testElement := DINT#100;
	fbAnyBuffer.PushRight(element := testElement);
	testElement := DINT#200;
	fbAnyBuffer.PushRight(element := testElement);

	// Act - Try to insert beyond elementCount
	testElement := DINT#999;
	Success := fbAnyBuffer.PushAtIndex(index := TEST_LL+3, element := testElement);  // elementCount = 2

	// Assert
	TestSuite.Test(__POUNAME()).AssertEqual(TEST_BOOL_FALSE, Success);
	TEST_DINT := 2;
	TestSuite.Test(__POUNAME()).AssertEqual(TEST_DINT, fbAnyBuffer.Metadata.elementCount);

	// Try index much larger than element count
	Success := fbAnyBuffer.PushAtIndex(index := TEST_UL+100, element := testElement);
	TestSuite.Test(__POUNAME()).AssertEqual(TEST_BOOL_FALSE, Success);
END_IF
END_METHOD

// FALSE returned for negative index
METHOD ReturnsFalseOnNegativeIndex
IF TestSuite.Test(__POUNAME()).ExecuteTest() THEN
	// Arrange
	fbAnyBuffer.Clear();
	testElement := DINT#100;
	fbAnyBuffer.PushRight(element := testElement);

	// Act
	testElement := DINT#999;
	Success := fbAnyBuffer.PushAtIndex(index := TEST_LL-1, element := testElement);

	// Assert
	TestSuite.Test(__POUNAME()).AssertEqual(TEST_BOOL_FALSE, Success);
	TEST_DINT := 1;
	TestSuite.Test(__POUNAME()).AssertEqual(TEST_DINT, fbAnyBuffer.Metadata.elementCount);
	TEST_DINT := 100;
	TestSuite.Test(__POUNAME()).AssertEqual(TEST_DINT, RawBuffer[TEST_LL+0]);
END_IF
END_METHOD

// Method returns TRUE when insert succeeds
METHOD ReturnsTrueOnSuccess
IF TestSuite.Test(__POUNAME()).ExecuteTest() THEN
	// Arrange
	fbAnyBuffer.Clear();
	testElement := DINT#100;
	fbAnyBuffer.PushRight(element := testElement);
	testElement := DINT#200;
	fbAnyBuffer.PushRight(element := testElement);

	// Act
	testElement := DINT#150;
	Success := fbAnyBuffer.PushAtIndex(index := TEST_LL+1, element := testElement);

	// Assert
	TestSuite.Test(__POUNAME()).AssertEqual(TEST_BOOL_TRUE, Success);
END_IF
END_METHOD

// All elements from index onward shift right by one
METHOD ShiftsElementsCorrectly
IF TestSuite.Test(__POUNAME()).ExecuteTest() THEN
	// Arrange - [100, 200, 300, 400]
	fbAnyBuffer.Clear();
	testElement := DINT#100;
	fbAnyBuffer.PushRight(element := testElement);
	testElement := DINT#200;
	fbAnyBuffer.PushRight(element := testElement);
	testElement := DINT#300;
	fbAnyBuffer.PushRight(element := testElement);
	testElement := DINT#400;
	fbAnyBuffer.PushRight(element := testElement);

	// Act - Insert 250 at index 2
	testElement := DINT#250;
	Success := fbAnyBuffer.PushAtIndex(index := TEST_LL+2, element := testElement);

	// Assert - [100, 200, 250, 300, 400]
	// Elements at index 2 and beyond shifted right: 300->index3, 400->index4
	TestSuite.Test(__POUNAME()).AssertEqual(TEST_BOOL_TRUE, Success);
	TEST_DINT := 100;
	TestSuite.Test(__POUNAME()).AssertEqual(TEST_DINT, RawBuffer[TEST_LL+0]);  // unchanged
	TEST_DINT := 200;
	TestSuite.Test(__POUNAME()).AssertEqual(TEST_DINT, RawBuffer[TEST_LL+1]);  // unchanged
	TEST_DINT := 250;
	TestSuite.Test(__POUNAME()).AssertEqual(TEST_DINT, RawBuffer[TEST_LL+2]);  // new element
	TEST_DINT := 300;
	TestSuite.Test(__POUNAME()).AssertEqual(TEST_DINT, RawBuffer[TEST_LL+3]);  // shifted from index 2
	TEST_DINT := 400;
	TestSuite.Test(__POUNAME()).AssertEqual(TEST_DINT, RawBuffer[TEST_LL+4]);  // shifted from index 3
END_IF
END_METHOD

// FALSE returned when element size doesn't match
METHOD WrongElementSize
IF TestSuite.Test(__POUNAME()).ExecuteTest() THEN
	// Arrange
	fbAnyBuffer.Clear();
	testElement := DINT#100;
	fbAnyBuffer.PushRight(element := testElement);

	// Act - Try to insert with wrong element size
	Success := fbAnyBuffer.PushAtIndex(index := TEST_LL, element := WrongSizeElement);

	// Assert - Should fail (BYTE is 1 byte, DINT is 4 bytes)
	TestSuite.Test(__POUNAME()).AssertEqual(TEST_BOOL_FALSE, Success);

	// Verify buffer element count unchanged
	TEST_DINT := 1;
	TestSuite.Test(__POUNAME()).AssertEqual(TEST_DINT, fbAnyBuffer.Metadata.elementCount);
	TEST_DINT := 100;
	TestSuite.Test(__POUNAME()).AssertEqual(TEST_DINT, RawBuffer[TEST_LL]);
END_IF
END_METHOD

END_PROGRAM

// ---- UnitTests/AnyBuffer/TEST_AnyBuffer_PeekAtIndex.TcPOU
PROGRAM TEST_AnyBuffer_PeekAtIndex
VAR
	// Loop counter
	i						: DINT;
END_VAR

PeekFromBeginning();
PeekFromMiddle();
PeekFromEnd();
ReturnsTrueOnSuccess();
ReturnsFalseOnNegativeIndex();
ReturnsFalseOnIndexOutOfBounds();
ReturnsFalseOnEmptyBuffer();
WrongElementSize();
EmptyElement();
BufferUnchangedAfterPeek();
ElementCountUnchanged();
MultiplePeeksOnSameIndex();
PeekAllPositions();
ElementOrderUnchanged();
ConsecutivePeeks();

// Buffer contents unchanged after peek
METHOD BufferUnchangedAfterPeek
IF TestSuite.Test(__POUNAME()).ExecuteTest() THEN
	// Arrange
	fbAnyBuffer.Clear();
	testElement := DINT#100;
	fbAnyBuffer.PushRight(element := testElement);
	testElement := DINT#200;
	fbAnyBuffer.PushRight(element := testElement);
	testElement := DINT#300;
	fbAnyBuffer.PushRight(element := testElement);

	// Act - Peek middle element
	Success := fbAnyBuffer.PeekAtIndex(index := TEST_LL+1, element := ReturnedElement);

	// Assert - Buffer should be unchanged
	TestSuite.Test(__POUNAME()).AssertEqual(TEST_BOOL_TRUE, Success);
	TEST_DINT := 200;
	TestSuite.Test(__POUNAME()).AssertEqual(TEST_DINT, ReturnedElement);

	// Verify all elements still in place
	TEST_DINT := 100;
	TestSuite.Test(__POUNAME()).AssertEqual(TEST_DINT, RawBuffer[TEST_LL+0]);
	TEST_DINT := 200;
	TestSuite.Test(__POUNAME()).AssertEqual(TEST_DINT, RawBuffer[TEST_LL+1]);
	TEST_DINT := 300;
	TestSuite.Test(__POUNAME()).AssertEqual(TEST_DINT, RawBuffer[TEST_LL+2]);
	TEST_DINT := 3;
	TestSuite.Test(__POUNAME()).AssertEqual(TEST_DINT, fbAnyBuffer.Metadata.elementCount);
END_IF
END_METHOD

// Multiple consecutive peeks at different indices work correctly
METHOD ConsecutivePeeks
IF TestSuite.Test(__POUNAME()).ExecuteTest() THEN
	// Arrange
	fbAnyBuffer.Clear();
	FOR i := 1 TO TEST_UL-TEST_LL+1 DO
		testElement := TO_DINT(i * 100);
		fbAnyBuffer.PushRight(element := testElement);
	END_FOR

	// Act - Peek multiple positions
	Success := fbAnyBuffer.PeekAtIndex(index := TEST_LL, element := ReturnedElement);
	TestSuite.Test(__POUNAME()).AssertEqual(TEST_BOOL_TRUE, Success);
	TEST_DINT := 100;
	TestSuite.Test(__POUNAME()).AssertEqual(TEST_DINT, ReturnedElement);

	Success := fbAnyBuffer.PeekAtIndex(index := TEST_LL+2, element := ReturnedElement);
	TestSuite.Test(__POUNAME()).AssertEqual(TEST_BOOL_TRUE, Success);
	TEST_DINT := 300;
	TestSuite.Test(__POUNAME()).AssertEqual(TEST_DINT, ReturnedElement);

	Success := fbAnyBuffer.PeekAtIndex(index := TEST_LL+4, element := ReturnedElement);
	TestSuite.Test(__POUNAME()).AssertEqual(TEST_BOOL_TRUE, Success);
	TEST_DINT := 500;
	TestSuite.Test(__POUNAME()).AssertEqual(TEST_DINT, ReturnedElement);

	// Assert - Buffer unchanged after all peeks
	TEST_DINT := 5;
	TestSuite.Test(__POUNAME()).AssertEqual(TEST_DINT, fbAnyBuffer.Metadata.elementCount);
	TEST_DINT := 100;
	TestSuite.Test(__POUNAME()).AssertEqual(TEST_DINT, RawBuffer[TEST_LL]);
	TEST_DINT := 500;
	TestSuite.Test(__POUNAME()).AssertEqual(TEST_DINT, RawBuffer[TEST_LL+4]);
END_IF
END_METHOD

// Element count remains same after peek
METHOD ElementCountUnchanged
IF TestSuite.Test(__POUNAME()).ExecuteTest() THEN
	// Arrange
	fbAnyBuffer.Clear();
	FOR i := 1 TO TEST_UL-TEST_LL+1 DO
		testElement := TO_DINT(i * 100);
		fbAnyBuffer.PushRight(element := testElement);
	END_FOR
	TEST_DINT := 5;
	TestSuite.Test(__POUNAME()).AssertEqual(TEST_DINT, fbAnyBuffer.Metadata.elementCount);

	// Act - Peek several times
	Success := fbAnyBuffer.PeekAtIndex(index := TEST_LL, element := ReturnedElement);
	TestSuite.Test(__POUNAME()).AssertEqual(TEST_BOOL_TRUE, Success);

	Success := fbAnyBuffer.PeekAtIndex(index := TEST_LL+2, element := ReturnedElement);
	TestSuite.Test(__POUNAME()).AssertEqual(TEST_BOOL_TRUE, Success);

	Success := fbAnyBuffer.PeekAtIndex(index := TEST_LL+4, element := ReturnedElement);
	TestSuite.Test(__POUNAME()).AssertEqual(TEST_BOOL_TRUE, Success);

	// Assert - Element count should be unchanged
	TEST_DINT := 5;
	TestSuite.Test(__POUNAME()).AssertEqual(TEST_DINT, fbAnyBuffer.Metadata.elementCount);
END_IF
END_METHOD

// Element order unchanged after multiple peeks
METHOD ElementOrderUnchanged
IF TestSuite.Test(__POUNAME()).ExecuteTest() THEN
	// Arrange - [100, 200, 300, 400, 500]
	fbAnyBuffer.Clear();
	FOR i := 1 TO TEST_UL-TEST_LL+1 DO
		testElement := TO_DINT(i * 100);
		fbAnyBuffer.PushRight(element := testElement);
	END_FOR

	// Act - Peek all elements in random order
	Success := fbAnyBuffer.PeekAtIndex(index := TEST_LL+2, element := ReturnedElement);
	Success := fbAnyBuffer.PeekAtIndex(index := TEST_LL+0, element := ReturnedElement);
	Success := fbAnyBuffer.PeekAtIndex(index := TEST_LL+4, element := ReturnedElement);
	Success := fbAnyBuffer.PeekAtIndex(index := TEST_LL+1, element := ReturnedElement);
	Success := fbAnyBuffer.PeekAtIndex(index := TEST_LL+3, element := ReturnedElement);

	// Assert - All elements should be in original positions
	TEST_DINT := 100;
	TestSuite.Test(__POUNAME()).AssertEqual(TEST_DINT, RawBuffer[TEST_LL+0]);
	TEST_DINT := 200;
	TestSuite.Test(__POUNAME()).AssertEqual(TEST_DINT, RawBuffer[TEST_LL+1]);
	TEST_DINT := 300;
	TestSuite.Test(__POUNAME()).AssertEqual(TEST_DINT, RawBuffer[TEST_LL+2]);
	TEST_DINT := 400;
	TestSuite.Test(__POUNAME()).AssertEqual(TEST_DINT, RawBuffer[TEST_LL+3]);
	TEST_DINT := 500;
	TestSuite.Test(__POUNAME()).AssertEqual(TEST_DINT, RawBuffer[TEST_LL+4]);
	TEST_DINT := 5;
	TestSuite.Test(__POUNAME()).AssertEqual(TEST_DINT, fbAnyBuffer.Metadata.elementCount);
END_IF
END_METHOD

// Behavior when element.diSize is 0 (validation only, no copy)
METHOD EmptyElement
VAR
	EmptyAny : __SYSTEM.AnyType;
END_VAR
IF TestSuite.Test(__POUNAME()).ExecuteTest() THEN
	// Arrange
	fbAnyBuffer.Clear();
	testElement := DINT#100;
	fbAnyBuffer.PushRight(element := testElement);
	testElement := DINT#200;
	fbAnyBuffer.PushRight(element := testElement);
	testElement := DINT#300;
	fbAnyBuffer.PushRight(element := testElement);

	// Act - Peek with empty element
	EmptyAny.diSize := 0;
	Success := fbAnyBuffer.PeekAtIndex(index := TEST_LL+1, element := EmptyAny);

	// Assert - Should fail
	TestSuite.Test(__POUNAME()).AssertEqual(TEST_BOOL_FALSE, Success);
	TEST_DINT := 3;
	TestSuite.Test(__POUNAME()).AssertEqual(TEST_DINT, fbAnyBuffer.Metadata.elementCount);
END_IF
END_METHOD

// Can peek same index multiple times with consistent results
METHOD MultiplePeeksOnSameIndex
IF TestSuite.Test(__POUNAME()).ExecuteTest() THEN
	// Arrange
	fbAnyBuffer.Clear();
	testElement := DINT#100;
	fbAnyBuffer.PushRight(element := testElement);
	testElement := DINT#200;
	fbAnyBuffer.PushRight(element := testElement);
	testElement := DINT#300;
	fbAnyBuffer.PushRight(element := testElement);

	// Act - Peek same index multiple times
	Success := fbAnyBuffer.PeekAtIndex(index := TEST_LL+1, element := ReturnedElement);
	TestSuite.Test(__POUNAME()).AssertEqual(TEST_BOOL_TRUE, Success);
	TEST_DINT := 200;
	TestSuite.Test(__POUNAME()).AssertEqual(TEST_DINT, ReturnedElement);

	Success := fbAnyBuffer.PeekAtIndex(index := TEST_LL+1, element := ReturnedElement);
	TestSuite.Test(__POUNAME()).AssertEqual(TEST_BOOL_TRUE, Success);
	TEST_DINT := 200;
	TestSuite.Test(__POUNAME()).AssertEqual(TEST_DINT, ReturnedElement);

	Success := fbAnyBuffer.PeekAtIndex(index := TEST_LL+1, element := ReturnedElement);
	TestSuite.Test(__POUNAME()).AssertEqual(TEST_BOOL_TRUE, Success);
	TEST_DINT := 200;
	TestSuite.Test(__POUNAME()).AssertEqual(TEST_DINT, ReturnedElement);

	// Assert - Buffer unchanged after multiple peeks
	TEST_DINT := 3;
	TestSuite.Test(__POUNAME()).AssertEqual(TEST_DINT, fbAnyBuffer.Metadata.elementCount);
END_IF
END_METHOD

// Can peek all valid positions in sequence
METHOD PeekAllPositions
IF TestSuite.Test(__POUNAME()).ExecuteTest() THEN
	// Arrange
	fbAnyBuffer.Clear();
	FOR i := 1 TO TEST_UL-TEST_LL+1 DO
		testElement := TO_DINT(i * 100);
		fbAnyBuffer.PushRight(element := testElement);
	END_FOR

	// Act & Assert - Peek all positions
	FOR i := TEST_LL TO TEST_UL DO
		Success := fbAnyBuffer.PeekAtIndex(index := TO_DINT(i), element := ReturnedElement);
		TestSuite.Test(__POUNAME()).AssertEqual(TEST_BOOL_TRUE, Success);
		TEST_DINT := TO_DINT((i - TEST_LL + 1) * 100);
		TestSuite.Test(__POUNAME()).AssertEqual(TEST_DINT, ReturnedElement);
	END_FOR

	// Assert - Buffer still full after peeking all positions
	TEST_DINT := TEST_UL-TEST_LL+1;
	TestSuite.Test(__POUNAME()).AssertEqual(TEST_DINT, fbAnyBuffer.Metadata.elementCount);
END_IF
END_METHOD

// Peeking at index 0 retrieves first element without modification
METHOD PeekFromBeginning
IF TestSuite.Test(__POUNAME()).ExecuteTest() THEN
	// Arrange
	fbAnyBuffer.Clear();
	testElement := DINT#100;
	fbAnyBuffer.PushRight(element := testElement);
	testElement := DINT#200;
	fbAnyBuffer.PushRight(element := testElement);
	testElement := DINT#300;
	fbAnyBuffer.PushRight(element := testElement);

	// Act
	Success := fbAnyBuffer.PeekAtIndex(index := TEST_LL, element := ReturnedElement);

	// Assert
	TestSuite.Test(__POUNAME()).AssertEqual(TEST_BOOL_TRUE, Success);
	TEST_DINT := 100;
	TestSuite.Test(__POUNAME()).AssertEqual(TEST_DINT, ReturnedElement);

	// Verify buffer unchanged
	TEST_DINT := 100;
	TestSuite.Test(__POUNAME()).AssertEqual(TEST_DINT, RawBuffer[TEST_LL+0]);
	TEST_DINT := 200;
	TestSuite.Test(__POUNAME()).AssertEqual(TEST_DINT, RawBuffer[TEST_LL+1]);
	TEST_DINT := 300;
	TestSuite.Test(__POUNAME()).AssertEqual(TEST_DINT, RawBuffer[TEST_LL+2]);
	TEST_DINT := 3;
	TestSuite.Test(__POUNAME()).AssertEqual(TEST_DINT, fbAnyBuffer.Metadata.elementCount);
END_IF
END_METHOD

// Peeking at last index retrieves last element
METHOD PeekFromEnd
IF TestSuite.Test(__POUNAME()).ExecuteTest() THEN
	// Arrange
	fbAnyBuffer.Clear();
	testElement := DINT#100;
	fbAnyBuffer.PushRight(element := testElement);
	testElement := DINT#200;
	fbAnyBuffer.PushRight(element := testElement);
	testElement := DINT#300;
	fbAnyBuffer.PushRight(element := testElement);

	// Act - Peek last element
	Success := fbAnyBuffer.PeekAtIndex(index := TEST_LL+2, element := ReturnedElement);

	// Assert
	TestSuite.Test(__POUNAME()).AssertEqual(TEST_BOOL_TRUE, Success);
	TEST_DINT := 300;
	TestSuite.Test(__POUNAME()).AssertEqual(TEST_DINT, ReturnedElement);

	// Verify buffer unchanged
	TEST_DINT := 100;
	TestSuite.Test(__POUNAME()).AssertEqual(TEST_DINT, RawBuffer[TEST_LL+0]);
	TEST_DINT := 200;
	TestSuite.Test(__POUNAME()).AssertEqual(TEST_DINT, RawBuffer[TEST_LL+1]);
	TEST_DINT := 300;
	TestSuite.Test(__POUNAME()).AssertEqual(TEST_DINT, RawBuffer[TEST_LL+2]);
	TEST_DINT := 3;
	TestSuite.Test(__POUNAME()).AssertEqual(TEST_DINT, fbAnyBuffer.Metadata.elementCount);
END_IF
END_METHOD

// Peeking from middle index retrieves correct element
METHOD PeekFromMiddle
IF TestSuite.Test(__POUNAME()).ExecuteTest() THEN
	// Arrange
	fbAnyBuffer.Clear();
	testElement := DINT#100;
	fbAnyBuffer.PushRight(element := testElement);
	testElement := DINT#200;
	fbAnyBuffer.PushRight(element := testElement);
	testElement := DINT#300;
	fbAnyBuffer.PushRight(element := testElement);
	testElement := DINT#400;
	fbAnyBuffer.PushRight(element := testElement);

	// Act - Peek middle element (index 1)
	Success := fbAnyBuffer.PeekAtIndex(index := TEST_LL+1, element := ReturnedElement);

	// Assert
	TestSuite.Test(__POUNAME()).AssertEqual(TEST_BOOL_TRUE, Success);
	TEST_DINT := 200;
	TestSuite.Test(__POUNAME()).AssertEqual(TEST_DINT, ReturnedElement);

	// Verify buffer unchanged
	TEST_DINT := 100;
	TestSuite.Test(__POUNAME()).AssertEqual(TEST_DINT, RawBuffer[TEST_LL]);
	TEST_DINT := 200;
	TestSuite.Test(__POUNAME()).AssertEqual(TEST_DINT, RawBuffer[TEST_LL+1]);
	TEST_DINT := 300;
	TestSuite.Test(__POUNAME()).AssertEqual(TEST_DINT, RawBuffer[TEST_LL+2]);
	TEST_DINT := 400;
	TestSuite.Test(__POUNAME()).AssertEqual(TEST_DINT, RawBuffer[TEST_LL+3]);
	TEST_DINT := 4;
	TestSuite.Test(__POUNAME()).AssertEqual(TEST_DINT, fbAnyBuffer.Metadata.elementCount);
END_IF
END_METHOD

// FALSE returned when buffer is empty (elementCount = 0)
METHOD ReturnsFalseOnEmptyBuffer
IF TestSuite.Test(__POUNAME()).ExecuteTest() THEN
	// Arrange
	fbAnyBuffer.Clear();

	// Act
	Success := fbAnyBuffer.PeekAtIndex(index := TEST_LL, element := ReturnedElement);

	// Assert
	TestSuite.Test(__POUNAME()).AssertEqual(TEST_BOOL_FALSE, Success);
	TEST_DINT := 0;
	TestSuite.Test(__POUNAME()).AssertEqual(TEST_DINT, fbAnyBuffer.Metadata.elementCount);
END_IF
END_METHOD

// FALSE returned when index >= elementCount
METHOD ReturnsFalseOnIndexOutOfBounds
IF TestSuite.Test(__POUNAME()).ExecuteTest() THEN
	// Arrange
	fbAnyBuffer.Clear();
	testElement := DINT#100;
	fbAnyBuffer.PushRight(element := testElement);
	testElement := DINT#200;
	fbAnyBuffer.PushRight(element := testElement);

	// Act - Try to peek beyond element count
	Success := fbAnyBuffer.PeekAtIndex(index := TEST_UL+1, element := ReturnedElement);

	// Assert
	TestSuite.Test(__POUNAME()).AssertEqual(TEST_BOOL_FALSE, Success);
	TEST_DINT := 2;
	TestSuite.Test(__POUNAME()).AssertEqual(TEST_DINT, fbAnyBuffer.Metadata.elementCount);

	// Try index much larger than element count
	Success := fbAnyBuffer.PeekAtIndex(index := TEST_UL+100, element := ReturnedElement);
	TestSuite.Test(__POUNAME()).AssertEqual(TEST_BOOL_FALSE, Success);
END_IF
END_METHOD

// FALSE returned for negative index
METHOD ReturnsFalseOnNegativeIndex
IF TestSuite.Test(__POUNAME()).ExecuteTest() THEN
	// Arrange
	fbAnyBuffer.Clear();
	testElement := DINT#100;
	fbAnyBuffer.PushRight(element := testElement);

	// Act
	Success := fbAnyBuffer.PeekAtIndex(index := TEST_LL-1, element := ReturnedElement);

	// Assert
	TestSuite.Test(__POUNAME()).AssertEqual(TEST_BOOL_FALSE, Success);
	TEST_DINT := 1;
	TestSuite.Test(__POUNAME()).AssertEqual(TEST_DINT, fbAnyBuffer.Metadata.elementCount);
END_IF
END_METHOD

// Method returns TRUE when peek succeeds
METHOD ReturnsTrueOnSuccess
IF TestSuite.Test(__POUNAME()).ExecuteTest() THEN
	// Arrange
	fbAnyBuffer.Clear();
	testElement := DINT#100;
	fbAnyBuffer.PushRight(element := testElement);
	testElement := DINT#200;
	fbAnyBuffer.PushRight(element := testElement);

	// Act
	Success := fbAnyBuffer.PeekAtIndex(index := TEST_LL, element := ReturnedElement);

	// Assert
	TestSuite.Test(__POUNAME()).AssertEqual(TEST_BOOL_TRUE, Success);
END_IF
END_METHOD

// FALSE returned when element size doesn't match
METHOD WrongElementSize
IF TestSuite.Test(__POUNAME()).ExecuteTest() THEN
	// Arrange
	fbAnyBuffer.Clear();
	testElement := DINT#100;
	fbAnyBuffer.PushRight(element := testElement);

	// Act - Try to peek with wrong element size
	Success := fbAnyBuffer.PeekAtIndex(index := TEST_LL, element := WrongSizeElement);

	// Assert - Should fail because of size difference
	TestSuite.Test(__POUNAME()).AssertEqual(TEST_BOOL_FALSE, Success);

	// Verify buffer unchanged
	TEST_DINT := 1;
	TestSuite.Test(__POUNAME()).AssertEqual(TEST_DINT, fbAnyBuffer.Metadata.elementCount);
	TEST_DINT := 100;
	TestSuite.Test(__POUNAME()).AssertEqual(TEST_DINT, RawBuffer[TEST_LL]);
END_IF
END_METHOD

END_PROGRAM

// ---- UnitTests/AnyBuffer/TEST_AnyBuffer_PopAtIndex.TcPOU
PROGRAM TEST_AnyBuffer_PopAtIndex
VAR
	// Loop counter
	i						: DINT;
END_VAR

PopFromBeginning();
PopFromMiddle();
PopFromEnd();
ReturnsTrueOnSuccess();
ReturnsFalseOnNegativeIndex();
ReturnsFalseOnIndexOutOfBounds();
ReturnsFalseOnEmptyBuffer();
WrongElementSize();
EmptyElement();
ShiftsElementsCorrectly();
ClearsLastPosition();
DecrementsElementCount();
ConsecutivePops();
PopAllElements();
ElementOrderPreserved();
PopAtIndexEquivalentToPopLeft();
PopAtIndexEquivalentToPopRight();

// The last position is cleared to zero after shift
METHOD ClearsLastPosition
IF TestSuite.Test(__POUNAME()).ExecuteTest() THEN
	// Arrange
	fbAnyBuffer.Clear();
	testElement := DINT#100;
	fbAnyBuffer.PushRight(element := testElement);
	testElement := DINT#200;
	fbAnyBuffer.PushRight(element := testElement);
	testElement := DINT#300;
	fbAnyBuffer.PushRight(element := testElement);

	// Act - Pop middle element
	Success := fbAnyBuffer.PopAtIndex(index := TEST_LL+1, element := ReturnedElement);

	// Assert - Last position should be cleared
	TestSuite.Test(__POUNAME()).AssertEqual(TEST_BOOL_TRUE, Success);
	TEST_DINT := 0;
	TestSuite.Test(__POUNAME()).AssertEqual(TEST_DINT, RawBuffer[TEST_LL+2]); // Position 2 was position 3, now cleared
END_IF
END_METHOD

// Multiple consecutive PopAtIndex calls maintain correct state
METHOD ConsecutivePops
IF TestSuite.Test(__POUNAME()).ExecuteTest() THEN
	// Arrange
	fbAnyBuffer.Clear();
	FOR i := 1 TO TEST_UL-TEST_LL+1 DO
		testElement := TO_DINT(i * 100);
		fbAnyBuffer.PushRight(element := testElement);
	END_FOR

	// Act - Pop multiple times at different indices
	Success := fbAnyBuffer.PopAtIndex(index := TEST_LL+2, element := ReturnedElement);  // Pop 300
	TestSuite.Test(__POUNAME()).AssertEqual(TEST_BOOL_TRUE, Success);
	TEST_DINT := 300;
	TestSuite.Test(__POUNAME()).AssertEqual(TEST_DINT, ReturnedElement);

	Success := fbAnyBuffer.PopAtIndex(index := TEST_LL+1, element := ReturnedElement);  // Pop 200
	TestSuite.Test(__POUNAME()).AssertEqual(TEST_BOOL_TRUE, Success);
	TEST_DINT := 200;
	TestSuite.Test(__POUNAME()).AssertEqual(TEST_DINT, ReturnedElement);

	Success := fbAnyBuffer.PopAtIndex(index := TEST_LL, element := ReturnedElement);  // Pop 100
	TestSuite.Test(__POUNAME()).AssertEqual(TEST_BOOL_TRUE, Success);
	TEST_DINT := 100;
	TestSuite.Test(__POUNAME()).AssertEqual(TEST_DINT, ReturnedElement);

	// Assert - Buffer should be [400, 500]
	TEST_DINT := 400;
	TestSuite.Test(__POUNAME()).AssertEqual(TEST_DINT, RawBuffer[TEST_LL]);
	TEST_DINT := 500;
	TestSuite.Test(__POUNAME()).AssertEqual(TEST_DINT, RawBuffer[TEST_LL+1]);
	TEST_DINT := 2;
	TestSuite.Test(__POUNAME()).AssertEqual(TEST_DINT, fbAnyBuffer.Metadata.elementCount);
END_IF
END_METHOD

// Element count decreases by 1 after pop
METHOD DecrementsElementCount
IF TestSuite.Test(__POUNAME()).ExecuteTest() THEN
	// Arrange
	fbAnyBuffer.Clear();
	FOR i := 1 TO 5 DO
		testElement := TO_DINT(i * 100);
		fbAnyBuffer.PushRight(element := testElement);
	END_FOR
	TEST_DINT := 5;
	TestSuite.Test(__POUNAME()).AssertEqual(TEST_DINT, fbAnyBuffer.Metadata.elementCount);

	// Act
	Success := fbAnyBuffer.PopAtIndex(index := TEST_LL+2, element := ReturnedElement);

	// Assert
	TestSuite.Test(__POUNAME()).AssertEqual(TEST_BOOL_TRUE, Success);
	TEST_DINT := 4;
	TestSuite.Test(__POUNAME()).AssertEqual(TEST_DINT, fbAnyBuffer.Metadata.elementCount);
END_IF
END_METHOD

// Element order is preserved after pop (except removed element)
METHOD ElementOrderPreserved
IF TestSuite.Test(__POUNAME()).ExecuteTest() THEN
	// Arrange - [100, 200, 300, 400, 500]
	fbAnyBuffer.Clear();
	FOR i := 1 TO 5 DO
		testElement := TO_DINT(i * 100);
		fbAnyBuffer.PushRight(element := testElement);
	END_FOR

	// Act - Remove 300 from middle
	Success := fbAnyBuffer.PopAtIndex(index := TEST_LL+2, element := ReturnedElement);

	// Assert - Order should be [100, 200, 400, 500]
	TestSuite.Test(__POUNAME()).AssertEqual(TEST_BOOL_TRUE, Success);
	TEST_DINT := 300;
	TestSuite.Test(__POUNAME()).AssertEqual(TEST_DINT, ReturnedElement);

	TEST_DINT := 100;
	TestSuite.Test(__POUNAME()).AssertEqual(TEST_DINT, RawBuffer[TEST_LL]);
	TEST_DINT := 200;
	TestSuite.Test(__POUNAME()).AssertEqual(TEST_DINT, RawBuffer[TEST_LL+1]);
	TEST_DINT := 400;
	TestSuite.Test(__POUNAME()).AssertEqual(TEST_DINT, RawBuffer[TEST_LL+2]);
	TEST_DINT := 500;
	TestSuite.Test(__POUNAME()).AssertEqual(TEST_DINT, RawBuffer[TEST_LL+3]);
END_IF
END_METHOD

// Behavior when element.diSize is 0 (discard mode)
METHOD EmptyElement
VAR
	EmptyAny : BYTE;
END_VAR
IF TestSuite.Test(__POUNAME()).ExecuteTest() THEN
	// Arrange
	fbAnyBuffer.Clear();
	testElement := DINT#100;
	fbAnyBuffer.PushRight(element := testElement);
	testElement := DINT#200;
	fbAnyBuffer.PushRight(element := testElement);
	testElement := DINT#300;
	fbAnyBuffer.PushRight(element := testElement);

	// Act - Pop but discard
	Success := fbAnyBuffer.PopAtIndex(index := TEST_LL+1, element := EmptyAny, TRUE);

	// Assert - Should succeed, element removed but not copied
	TestSuite.Test(__POUNAME()).AssertEqual(TEST_BOOL_TRUE, Success);
	TEST_DINT := 2;
	TestSuite.Test(__POUNAME()).AssertEqual(TEST_DINT, fbAnyBuffer.Metadata.elementCount);
	TEST_DINT := 100;
	TestSuite.Test(__POUNAME()).AssertEqual(TEST_DINT, RawBuffer[TEST_LL+0]);
	TEST_DINT := 300;
	TestSuite.Test(__POUNAME()).AssertEqual(TEST_DINT, RawBuffer[TEST_LL+1]);
END_IF
END_METHOD

// Can pop all elements sequentially using index 0
METHOD PopAllElements
IF TestSuite.Test(__POUNAME()).ExecuteTest() THEN
	// Arrange
	fbAnyBuffer.Clear();
	FOR i := 1 TO TEST_UL-TEST_LL+1 DO
		testElement := TO_DINT(i * 100);
		fbAnyBuffer.PushRight(element := testElement);
	END_FOR

	// Act - Pop all elements from index 0
	FOR i := 1 TO TEST_UL-TEST_LL+1 DO
		Success := fbAnyBuffer.PopAtIndex(index := TEST_LL, element := ReturnedElement);
		TestSuite.Test(__POUNAME()).AssertEqual(TEST_BOOL_TRUE, Success);
		TEST_DINT := TO_DINT(i * 100);
		TestSuite.Test(__POUNAME()).AssertEqual(TEST_DINT, ReturnedElement);
	END_FOR

	// Assert - Buffer should be empty
	TEST_DINT := 0;
	TestSuite.Test(__POUNAME()).AssertEqual(TEST_DINT, fbAnyBuffer.Metadata.elementCount);
END_IF
END_METHOD

// PopAtIndex(0) behaves same as PopLeft
METHOD PopAtIndexEquivalentToPopLeft
VAR
	popLeftValue : DINT;
	popAtIndexValue : DINT;
END_VAR
IF TestSuite.Test(__POUNAME()).ExecuteTest() THEN
	// Arrange - Two identical buffers
	fbAnyBuffer.Clear();
	FOR i := 1 TO 5 DO
		testElement := TO_DINT(i * 100);
		fbAnyBuffer.PushRight(element := testElement);
	END_FOR

	// Act - Pop using PopLeft
	Success := fbAnyBuffer.PopLeft(element := popLeftValue);
	TestSuite.Test(__POUNAME()).AssertEqual(TEST_BOOL_TRUE, Success);

	// Clear and rebuild buffer
	fbAnyBuffer.Clear();
	FOR i := 1 TO TEST_UL-TEST_LL+1 DO
		testElement := TO_DINT(i * 100);
		fbAnyBuffer.PushRight(element := testElement);
	END_FOR

	// Act - Pop using PopAtIndex(TEST_LL)
	Success := fbAnyBuffer.PopAtIndex(index := TEST_LL, element := popAtIndexValue);
	TestSuite.Test(__POUNAME()).AssertEqual(TEST_BOOL_TRUE, Success);

	// Assert - Both should return same value
	TestSuite.Test(__POUNAME()).AssertEqual(popLeftValue, popAtIndexValue);
	TEST_DINT := 100;
	TestSuite.Test(__POUNAME()).AssertEqual(TEST_DINT, popAtIndexValue);
END_IF
END_METHOD

// PopAtIndex(elementCount-1) behaves same as PopRight
METHOD PopAtIndexEquivalentToPopRight
VAR
	popRightValue : DINT;
	popAtIndexValue : DINT;
	lastIndex : DINT;
END_VAR
IF TestSuite.Test(__POUNAME()).ExecuteTest() THEN
	// Arrange - Two identical buffers
	fbAnyBuffer.Clear();
	FOR i := 1 TO 5 DO
		testElement := TO_DINT(i * 100);
		fbAnyBuffer.PushRight(element := testElement);
	END_FOR

	// Act - Pop using PopRight
	Success := fbAnyBuffer.PopRight(element := popRightValue);
	TestSuite.Test(__POUNAME()).AssertEqual(TEST_BOOL_TRUE, Success);

	// Clear and rebuild buffer
	fbAnyBuffer.Clear();
	FOR i := 1 TO 5 DO
		testElement := TO_DINT(i * 100);
		fbAnyBuffer.PushRight(element := testElement);
	END_FOR

	// Act - Pop using PopAtIndex(elementCount-1)
	lastIndex := fbAnyBuffer.Metadata.elementCount - 1;
	Success := fbAnyBuffer.PopAtIndex(index := TEST_LL+lastIndex, element := popAtIndexValue);
	TestSuite.Test(__POUNAME()).AssertEqual(TEST_BOOL_TRUE, Success);

	// Assert - Both should return same value
	TestSuite.Test(__POUNAME()).AssertEqual(popRightValue, popAtIndexValue);
	TEST_DINT := 500;
	TestSuite.Test(__POUNAME()).AssertEqual(TEST_DINT, popAtIndexValue);
END_IF
END_METHOD

// Popping at index 0 retrieves first element and shifts all
METHOD PopFromBeginning
IF TestSuite.Test(__POUNAME()).ExecuteTest() THEN
	// Arrange
	fbAnyBuffer.Clear();
	testElement := DINT#100;
	fbAnyBuffer.PushRight(element := testElement);
	testElement := DINT#200;
	fbAnyBuffer.PushRight(element := testElement);
	testElement := DINT#300;
	fbAnyBuffer.PushRight(element := testElement);

	// Act
	Success := fbAnyBuffer.PopAtIndex(index := TEST_LL, element := ReturnedElement);

	// Assert
	TestSuite.Test(__POUNAME()).AssertEqual(TEST_BOOL_TRUE, Success);
	TEST_DINT := 100;
	TestSuite.Test(__POUNAME()).AssertEqual(TEST_DINT, ReturnedElement);

	// Verify elements shifted left
	TEST_DINT := 200;
	TestSuite.Test(__POUNAME()).AssertEqual(TEST_DINT, RawBuffer[TEST_LL]);
	TEST_DINT := 300;
	TestSuite.Test(__POUNAME()).AssertEqual(TEST_DINT, RawBuffer[TEST_LL+1]);
	TEST_DINT := 2;
	TestSuite.Test(__POUNAME()).AssertEqual(TEST_DINT, fbAnyBuffer.Metadata.elementCount);
END_IF
END_METHOD

// Popping at last index (elementCount-1) retrieves last element
METHOD PopFromEnd
IF TestSuite.Test(__POUNAME()).ExecuteTest() THEN
	// Arrange
	fbAnyBuffer.Clear();
	testElement := DINT#100;
	fbAnyBuffer.PushRight(element := testElement);
	testElement := DINT#200;
	fbAnyBuffer.PushRight(element := testElement);
	testElement := DINT#300;
	fbAnyBuffer.PushRight(element := testElement);

	// Act - Pop last element
	Success := fbAnyBuffer.PopAtIndex(index := TEST_LL+2, element := ReturnedElement);

	// Assert
	TestSuite.Test(__POUNAME()).AssertEqual(TEST_BOOL_TRUE, Success);
	TEST_DINT := 300;
	TestSuite.Test(__POUNAME()).AssertEqual(TEST_DINT, ReturnedElement);

	// Verify remaining elements unchanged
	TEST_DINT := 100;
	TestSuite.Test(__POUNAME()).AssertEqual(TEST_DINT, RawBuffer[TEST_LL+0]);
	TEST_DINT := 200;
	TestSuite.Test(__POUNAME()).AssertEqual(TEST_DINT, RawBuffer[TEST_LL+1]);
	TEST_DINT := 2;
	TestSuite.Test(__POUNAME()).AssertEqual(TEST_DINT, fbAnyBuffer.Metadata.elementCount);
END_IF
END_METHOD

// Popping from middle index retrieves correct element and shifts remaining
METHOD PopFromMiddle
IF TestSuite.Test(__POUNAME()).ExecuteTest() THEN
	// Arrange
	fbAnyBuffer.Clear();
	testElement := DINT#100;
	fbAnyBuffer.PushRight(element := testElement);
	testElement := DINT#200;
	fbAnyBuffer.PushRight(element := testElement);
	testElement := DINT#300;
	fbAnyBuffer.PushRight(element := testElement);
	testElement := DINT#400;
	fbAnyBuffer.PushRight(element := testElement);

	// Act - Pop middle element (index 1)
	Success := fbAnyBuffer.PopAtIndex(index := TEST_LL+1, element := ReturnedElement);

	// Assert
	TestSuite.Test(__POUNAME()).AssertEqual(TEST_BOOL_TRUE, Success);
	TEST_DINT := 200;
	TestSuite.Test(__POUNAME()).AssertEqual(TEST_DINT, ReturnedElement);

	// Verify elements after index shifted left
	TEST_DINT := 100;
	TestSuite.Test(__POUNAME()).AssertEqual(TEST_DINT, RawBuffer[TEST_LL+0]);
	TEST_DINT := 300;
	TestSuite.Test(__POUNAME()).AssertEqual(TEST_DINT, RawBuffer[TEST_LL+1]);
	TEST_DINT := 400;
	TestSuite.Test(__POUNAME()).AssertEqual(TEST_DINT, RawBuffer[TEST_LL+2]);
	TEST_DINT := 3;
	TestSuite.Test(__POUNAME()).AssertEqual(TEST_DINT, fbAnyBuffer.Metadata.elementCount);
END_IF
END_METHOD

// FALSE returned when buffer is empty (elementCount = 0)
METHOD ReturnsFalseOnEmptyBuffer
IF TestSuite.Test(__POUNAME()).ExecuteTest() THEN
	// Arrange
	fbAnyBuffer.Clear();

	// Act
	Success := fbAnyBuffer.PopAtIndex(index := TEST_LL, element := ReturnedElement);

	// Assert
	TestSuite.Test(__POUNAME()).AssertEqual(TEST_BOOL_FALSE, Success);
	TEST_DINT := 0;
	TestSuite.Test(__POUNAME()).AssertEqual(TEST_DINT, fbAnyBuffer.Metadata.elementCount);
END_IF
END_METHOD

// FALSE returned when index >= elementCount
METHOD ReturnsFalseOnIndexOutOfBounds
IF TestSuite.Test(__POUNAME()).ExecuteTest() THEN
	// Arrange
	fbAnyBuffer.Clear();
	testElement := DINT#100;
	fbAnyBuffer.PushRight(element := testElement);
	testElement := DINT#200;
	fbAnyBuffer.PushRight(element := testElement);

	// Act - Try to pop beyond element count
	Success := fbAnyBuffer.PopAtIndex(index := TEST_LL+2, element := ReturnedElement);

	// Assert
	TestSuite.Test(__POUNAME()).AssertEqual(TEST_BOOL_FALSE, Success);
	TEST_DINT := 2;
	TestSuite.Test(__POUNAME()).AssertEqual(TEST_DINT, fbAnyBuffer.Metadata.elementCount);

	// Try index much larger than element count
	Success := fbAnyBuffer.PopAtIndex(index := TEST_UL+100, element := ReturnedElement);
	TestSuite.Test(__POUNAME()).AssertEqual(TEST_BOOL_FALSE, Success);
END_IF
END_METHOD

// FALSE returned for negative index
METHOD ReturnsFalseOnNegativeIndex
IF TestSuite.Test(__POUNAME()).ExecuteTest() THEN
	// Arrange
	fbAnyBuffer.Clear();
	testElement := DINT#100;
	fbAnyBuffer.PushRight(element := testElement);

	// Act
	Success := fbAnyBuffer.PopAtIndex(index := TEST_LL-1, element := ReturnedElement);

	// Assert
	TestSuite.Test(__POUNAME()).AssertEqual(TEST_BOOL_FALSE, Success);
	TEST_DINT := 1;
	TestSuite.Test(__POUNAME()).AssertEqual(TEST_DINT, fbAnyBuffer.Metadata.elementCount);
END_IF
END_METHOD

// Method returns TRUE when pop succeeds
METHOD ReturnsTrueOnSuccess
IF TestSuite.Test(__POUNAME()).ExecuteTest() THEN
	// Arrange
	fbAnyBuffer.Clear();
	testElement := DINT#100;
	fbAnyBuffer.PushRight(element := testElement);
	testElement := DINT#200;
	fbAnyBuffer.PushRight(element := testElement);

	// Act
	Success := fbAnyBuffer.PopAtIndex(index := TEST_LL, element := ReturnedElement);

	// Assert
	TestSuite.Test(__POUNAME()).AssertEqual(TEST_BOOL_TRUE, Success);
END_IF
END_METHOD

// All elements after index shift left by one position
METHOD ShiftsElementsCorrectly
IF TestSuite.Test(__POUNAME()).ExecuteTest() THEN
	// Arrange - [100, 200, 300, 400, 500]
	fbAnyBuffer.Clear();
	FOR i := 1 TO 5 DO
		testElement := TO_DINT(i * 100);
		fbAnyBuffer.PushRight(element := testElement);
	END_FOR

	// Act - Remove 200 (index 1)
	Success := fbAnyBuffer.PopAtIndex(index := TEST_LL+1, element := ReturnedElement);

	// Assert - Buffer should be [100, 300, 400, 500]
	TestSuite.Test(__POUNAME()).AssertEqual(TEST_BOOL_TRUE, Success);
	TEST_DINT := 200;
	TestSuite.Test(__POUNAME()).AssertEqual(TEST_DINT, ReturnedElement);

	// Verify all elements after index 1 shifted left
	TEST_DINT := 100;
	TestSuite.Test(__POUNAME()).AssertEqual(TEST_DINT, RawBuffer[TEST_LL+0]);
	TEST_DINT := 300;
	TestSuite.Test(__POUNAME()).AssertEqual(TEST_DINT, RawBuffer[TEST_LL+1]);  // Was at index 2
	TEST_DINT := 400;
	TestSuite.Test(__POUNAME()).AssertEqual(TEST_DINT, RawBuffer[TEST_LL+2]);  // Was at index 3
	TEST_DINT := 500;
	TestSuite.Test(__POUNAME()).AssertEqual(TEST_DINT, RawBuffer[TEST_LL+3]);  // Was at index 4
	TEST_DINT := 4;
	TestSuite.Test(__POUNAME()).AssertEqual(TEST_DINT, fbAnyBuffer.Metadata.elementCount);
END_IF
END_METHOD

// FALSE returned when element size doesn't match
METHOD WrongElementSize
IF TestSuite.Test(__POUNAME()).ExecuteTest() THEN
	// Arrange
	fbAnyBuffer.Clear();
	testElement := DINT#100;
	fbAnyBuffer.PushRight(element := testElement);

	// Act - Try to pop with wrong element size
	Success := fbAnyBuffer.PopAtIndex(index := TEST_LL, element := WrongSizeElement);

	// Assert - Should fail because of size difference
	TestSuite.Test(__POUNAME()).AssertEqual(TEST_BOOL_FALSE, Success);

	// Verify buffer unchanged
	TEST_DINT := 1;
	TestSuite.Test(__POUNAME()).AssertEqual(TEST_DINT, fbAnyBuffer.Metadata.elementCount);
	TEST_DINT := 100;
	TestSuite.Test(__POUNAME()).AssertEqual(TEST_DINT, RawBuffer[TEST_LL]);
END_IF
END_METHOD

END_PROGRAM

// ---- UnitTests/AnyBuffer/TEST_AnyBuffer_PopLeft.TcPOU
PROGRAM TEST_AnyBuffer_PopLeft
VAR
	// Loop counter
	i						: DINT;
END_VAR

RetrievesFirstElement();
ShiftsElements();
ClearsLastElement();
DecrementsElementCount();
ReturnsTrueOnSuccess();
WrongSize();
EmptyElement();
PopFromEmptyBuffer();
PopSingleElement();
ConsecutivePops();
PopAfterAppendLeft();
PopAfterAppendRight();
PopUntilEmpty();
ElementOrderPreserved();
PopDiscardTrue();
PopDiscardTrueSkipsTypeCheck();
PopDiscardTrueShiftsElements();
PopDiscardTrueDecrementsCount();
PopDiscardFalseRetrievesValue();
PopDiscardFalseValidatesType();
PopDiscardWithWrongTypeSucceeds();
PopDiscardReturnsTrueOnSuccess();

// PopLeft clears the last element of the buffer after shifting
METHOD ClearsLastElement
IF TestSuite.Test(__POUNAME()).ExecuteTest() THEN
	// Arrange
	fbAnyBuffer.Clear();
	RawBuffer[TEST_LL+0] := 100;
	RawBuffer[TEST_LL+1] := 200;
	RawBuffer[TEST_LL+2] := 300;
	RawBuffer[TEST_LL+3] := 400;
	RawBuffer[TEST_LL+4] := 500;
	fbAnyBuffer.Metadata.elementCount := 5;
	ReturnedElement := 0;

	// Act
	Success := fbAnyBuffer.PopLeft(element := ReturnedElement);

	// Assert - Last element should be cleared (0)
	TEST_DINT := 0;
	TestSuite.Test(__POUNAME()).AssertEqual(TEST_DINT, RawBuffer[TEST_LL+4]);
END_IF
END_METHOD

// PopLeft multiple times maintains correct order
METHOD ConsecutivePops
VAR
	pop1 : DINT;
	pop2 : DINT;
	pop3 : DINT;
END_VAR
IF TestSuite.Test(__POUNAME()).ExecuteTest() THEN
	// Arrange - Fill buffer with sequential values
	fbAnyBuffer.Clear();
	RawBuffer[TEST_LL+0] := 10;
	RawBuffer[TEST_LL+1] := 20;
	RawBuffer[TEST_LL+2] := 30;
	RawBuffer[TEST_LL+3] := 40;
	RawBuffer[TEST_LL+4] := 50;
	fbAnyBuffer.Metadata.elementCount := 5;

	// Act - Pop three times consecutively
	fbAnyBuffer.PopLeft(element := pop1);
	fbAnyBuffer.PopLeft(element := pop2);
	fbAnyBuffer.PopLeft(element := pop3);

	// Assert - Elements should be retrieved in FIFO order
	TEST_DINT := 10;
	TestSuite.Test(__POUNAME()).AssertEqual(TEST_DINT, pop1);
	TEST_DINT := 20;
	TestSuite.Test(__POUNAME()).AssertEqual(TEST_DINT, pop2);
	TEST_DINT := 30;
	TestSuite.Test(__POUNAME()).AssertEqual(TEST_DINT, pop3);

	// Remaining buffer state: [40, 50, 0, 0, 0]
	TEST_DINT := 40;
	TestSuite.Test(__POUNAME()).AssertEqual(TEST_DINT, RawBuffer[TEST_LL+0]);
	TEST_DINT := 50;
	TestSuite.Test(__POUNAME()).AssertEqual(TEST_DINT, RawBuffer[TEST_LL+1]);
	TEST_DINT := 0;
	TestSuite.Test(__POUNAME()).AssertEqual(TEST_DINT, RawBuffer[TEST_LL+2]);
	TestSuite.Test(__POUNAME()).AssertEqual(TEST_DINT, RawBuffer[TEST_LL+3]);
	TestSuite.Test(__POUNAME()).AssertEqual(TEST_DINT, RawBuffer[TEST_LL+4]);
END_IF
END_METHOD

// Element count decreases by 1 after pop
METHOD DecrementsElementCount
IF TestSuite.Test(__POUNAME()).ExecuteTest() THEN
	// Arrange
	fbAnyBuffer.Clear();
	RawBuffer[TEST_LL+0] := 100;
	RawBuffer[TEST_LL+1] := 200;
	RawBuffer[TEST_LL+2] := 300;
	fbAnyBuffer.Metadata.elementCount := 3;
	TEST_DINT := 3;
	TestSuite.Test(__POUNAME()).AssertEqual(TEST_DINT, fbAnyBuffer.Metadata.elementCount);

	// Act
	Success := fbAnyBuffer.PopLeft(element := ReturnedElement);

	// Assert
	TestSuite.Test(__POUNAME()).AssertEqual(TEST_BOOL_TRUE, Success);
	TEST_DINT := 2;
	TestSuite.Test(__POUNAME()).AssertEqual(TEST_DINT, fbAnyBuffer.Metadata.elementCount);
END_IF
END_METHOD

// Remaining elements shift correctly and maintain relative order
METHOD ElementOrderPreserved
VAR
	ReturnedElement : DINT;
END_VAR
IF TestSuite.Test(__POUNAME()).ExecuteTest() THEN
	// Arrange - [100, 200, 300, 400, 500]
	fbAnyBuffer.Clear();
	FOR i := 1 TO 5 DO
		AppendedElement := TO_DINT(i * 100);
		fbAnyBuffer.PushRight(AppendedElement);
	END_FOR

	// Act - Pop first element (100)
	Success := fbAnyBuffer.PopLeft(element := ReturnedElement);

	// Assert - Order should be [200, 300, 400, 500]
	TestSuite.Test(__POUNAME()).AssertEqual(TEST_BOOL_TRUE, Success);
	TEST_DINT := 100;
	TestSuite.Test(__POUNAME()).AssertEqual(TEST_DINT, ReturnedElement);

	TEST_DINT := 200;
	TestSuite.Test(__POUNAME()).AssertEqual(TEST_DINT, RawBuffer[TEST_LL+0]);
	TEST_DINT := 300;
	TestSuite.Test(__POUNAME()).AssertEqual(TEST_DINT, RawBuffer[TEST_LL+1]);
	TEST_DINT := 400;
	TestSuite.Test(__POUNAME()).AssertEqual(TEST_DINT, RawBuffer[TEST_LL+2]);
	TEST_DINT := 500;
	TestSuite.Test(__POUNAME()).AssertEqual(TEST_DINT, RawBuffer[TEST_LL+3]);
	TEST_DINT := 4;
	TestSuite.Test(__POUNAME()).AssertEqual(TEST_DINT, fbAnyBuffer.Metadata.elementCount);
END_IF
END_METHOD

// PopLeft with zero-sized element just shifts without copying
METHOD EmptyElement
VAR
	EmptyAny				: __SYSTEM.AnyType;
END_VAR
IF TestSuite.Test(__POUNAME()).ExecuteTest() THEN
	// Arrange
	fbAnyBuffer.Clear();
	RawBuffer[TEST_LL+0] := 100;
	RawBuffer[TEST_LL+1] := 200;
	RawBuffer[TEST_LL+2] := 300;
	fbAnyBuffer.Metadata.elementCount := 3;
	fbAnyBuffer.Metadata.capacity := 2;

	// Initialize empty AnyType (size = 0)
	EmptyAny.pValue := 0;
	EmptyAny.diSize := 0;

	// Act - Call with zero-sized element
	Success := fbAnyBuffer.PopLeft(element := EmptyAny);

	// Assert - Should NOT succeed and shift elements
	TestSuite.Test(__POUNAME()).AssertEqual(TEST_BOOL_FALSE, Success);
	TEST_DINT := 100;
	TestSuite.Test(__POUNAME()).AssertEqual(TEST_DINT, RawBuffer[TEST_LL+0]);
	TEST_DINT := 200;
	TestSuite.Test(__POUNAME()).AssertEqual(TEST_DINT, RawBuffer[TEST_LL+1]);
	TEST_DINT := 300;
	TestSuite.Test(__POUNAME()).AssertEqual(TEST_DINT, RawBuffer[TEST_LL+2]);
END_IF
END_METHOD

// AppendLeft and PopLeft demonstrate LIFO behavior
METHOD PopAfterAppendLeft
VAR
	ReturnedElement : DINT;
END_VAR
IF TestSuite.Test(__POUNAME()).ExecuteTest() THEN
	// Arrange
	fbAnyBuffer.Clear();

	// Act - Append then Pop (LIFO: Last In First Out)
	AppendedElement := DINT#100;
	fbAnyBuffer.PushLeft(element := AppendedElement);  // [100]
	AppendedElement := DINT#200;
	fbAnyBuffer.PushLeft(element := AppendedElement);  // [200, 100]
	AppendedElement := DINT#300;
	fbAnyBuffer.PushLeft(element := AppendedElement);  // [300, 200, 100]
	fbAnyBuffer.PopLeft(element := ReturnedElement);  // Pop 300

	// Assert - Should pop the last appended value (300)
	TEST_DINT := 300;
	TestSuite.Test(__POUNAME()).AssertEqual(TEST_DINT, ReturnedElement);

	// Buffer should now be [200, 100]
	TEST_DINT := 200;
	TestSuite.Test(__POUNAME()).AssertEqual(TEST_DINT, RawBuffer[TEST_LL+0]);
	TEST_DINT := 100;
	TestSuite.Test(__POUNAME()).AssertEqual(TEST_DINT, RawBuffer[TEST_LL+1]);
END_IF
END_METHOD

// AppendRight and PopLeft demonstrate FIFO behavior
METHOD PopAfterAppendRight
VAR
	ReturnedElement : DINT;
END_VAR
IF TestSuite.Test(__POUNAME()).ExecuteTest() THEN
	// Arrange
	fbAnyBuffer.Clear();

	// Act - Append Right and Pop Left (FIFO: First In First Out)
	AppendedElement := DINT#100;
	fbAnyBuffer.PushRight(element := AppendedElement);  // [100]
	AppendedElement := DINT#200;
	fbAnyBuffer.PushRight(element := AppendedElement);  // [100, 200]
	AppendedElement := DINT#300;
	fbAnyBuffer.PushRight(element := AppendedElement);  // [100, 200, 300]
	fbAnyBuffer.PopLeft(element := ReturnedElement);  // Pop 100 (first appended)

	// Assert - Should pop the first appended value (100)
	TEST_DINT := 100;
	TestSuite.Test(__POUNAME()).AssertEqual(TEST_DINT, ReturnedElement);

	// Buffer should now be [200, 300]
	TEST_DINT := 200;
	TestSuite.Test(__POUNAME()).AssertEqual(TEST_DINT, RawBuffer[TEST_LL+0]);
	TEST_DINT := 300;
	TestSuite.Test(__POUNAME()).AssertEqual(TEST_DINT, RawBuffer[TEST_LL+1]);
	TEST_DINT := 2;
	TestSuite.Test(__POUNAME()).AssertEqual(TEST_DINT, fbAnyBuffer.Metadata.elementCount);
END_IF
END_METHOD

// Element value is copied when popDiscard=FALSE (default)
METHOD PopDiscardFalseRetrievesValue
IF TestSuite.Test(__POUNAME()).ExecuteTest() THEN
	// Arrange
	fbAnyBuffer.Clear();
	RawBuffer[TEST_LL+0] := 123;
	RawBuffer[TEST_LL+1] := 456;
	fbAnyBuffer.Metadata.elementCount := 2;
	ReturnedElement := 0;

	// Act - Pop with explicit popDiscard=FALSE
	Success := fbAnyBuffer.PopLeft(element := ReturnedElement, popDiscard := FALSE);

	// Assert - Value is retrieved
	TestSuite.Test(__POUNAME()).AssertEqual(TEST_BOOL_TRUE, Success);
	TEST_DINT := 123;
	TestSuite.Test(__POUNAME()).AssertEqual(TEST_DINT, ReturnedElement);
END_IF
END_METHOD

// Type checking occurs when popDiscard=FALSE
METHOD PopDiscardFalseValidatesType
IF TestSuite.Test(__POUNAME()).ExecuteTest() THEN
	// Arrange
	fbAnyBuffer.Clear();
	RawBuffer[TEST_LL+0] := 100;
	fbAnyBuffer.Metadata.elementCount := 1;
	WrongSizeElement := 0;

	// Act - Pop with wrong type and popDiscard=FALSE (should fail)
	Success := fbAnyBuffer.PopLeft(element := WrongSizeElement, popDiscard := FALSE);

	// Assert - Should fail due to type mismatch
	TestSuite.Test(__POUNAME()).AssertEqual(TEST_BOOL_FALSE, Success);
	// Element count should remain unchanged (pop failed)
	TEST_DINT := 1;
	TestSuite.Test(__POUNAME()).AssertEqual(TEST_DINT, fbAnyBuffer.Metadata.elementCount);
END_IF
END_METHOD

// Method returns TRUE when popDiscard=TRUE succeeds
METHOD PopDiscardReturnsTrueOnSuccess
VAR
	discardBuffer : DINT;
END_VAR
IF TestSuite.Test(__POUNAME()).ExecuteTest() THEN
	// Arrange
	fbAnyBuffer.Clear();
	RawBuffer[TEST_LL+0] := 777;
	fbAnyBuffer.Metadata.elementCount := 1;

	// Act
	Success := fbAnyBuffer.PopLeft(element := discardBuffer, popDiscard := TRUE);

	// Assert
	TestSuite.Test(__POUNAME()).AssertEqual(TEST_BOOL_TRUE, Success);
	TEST_DINT := 0;  // Buffer empty
	TestSuite.Test(__POUNAME()).AssertEqual(TEST_DINT, fbAnyBuffer.Metadata.elementCount);
END_IF
END_METHOD

// Element is removed but not copied when popDiscard=TRUE
METHOD PopDiscardTrue
VAR
	discardBuffer : BYTE;  // Can be any type when popDiscard=TRUE
END_VAR
IF TestSuite.Test(__POUNAME()).ExecuteTest() THEN
	// Arrange
	fbAnyBuffer.Clear();
	RawBuffer[TEST_LL+0] := 100;
	RawBuffer[TEST_LL+1] := 200;
	RawBuffer[TEST_LL+2] := 300;
	fbAnyBuffer.Metadata.elementCount := 3;
	discardBuffer := 0;

	// Act - Pop with discard=TRUE
	Success := fbAnyBuffer.PopLeft(element := discardBuffer, popDiscard := TRUE);

	// Assert - Success but discardBuffer unchanged (no copy occurred)
	TestSuite.Test(__POUNAME()).AssertEqual(TEST_BOOL_TRUE, Success);
	TEST_DINT := 2;
	TestSuite.Test(__POUNAME()).AssertEqual(TEST_DINT, fbAnyBuffer.Metadata.elementCount);
	// Buffer should be shifted: [200, 300, 0]
	TEST_DINT := 200;
	TestSuite.Test(__POUNAME()).AssertEqual(TEST_DINT, RawBuffer[TEST_LL+0]);
	TEST_DINT := 300;
	TestSuite.Test(__POUNAME()).AssertEqual(TEST_DINT, RawBuffer[TEST_LL+1]);
END_IF
END_METHOD

// ElementCount decreases when popDiscard=TRUE
METHOD PopDiscardTrueDecrementsCount
VAR
	discardBuffer : DINT;
END_VAR
IF TestSuite.Test(__POUNAME()).ExecuteTest() THEN
	// Arrange
	fbAnyBuffer.Clear();
	RawBuffer[TEST_LL+0] := 100;
	RawBuffer[TEST_LL+1] := 200;
	RawBuffer[TEST_LL+2] := 300;
	fbAnyBuffer.Metadata.elementCount := 3;
	TEST_DINT := 3;
	TestSuite.Test(__POUNAME()).AssertEqual(TEST_DINT, fbAnyBuffer.Metadata.elementCount);

	// Act - Pop with discard=TRUE
	Success := fbAnyBuffer.PopLeft(element := discardBuffer, popDiscard := TRUE);

	// Assert - Count decremented
	TestSuite.Test(__POUNAME()).AssertEqual(TEST_BOOL_TRUE, Success);
	TEST_DINT := 2;
	TestSuite.Test(__POUNAME()).AssertEqual(TEST_DINT, fbAnyBuffer.Metadata.elementCount);
END_IF
END_METHOD

// Elements still shift correctly when popDiscard=TRUE
METHOD PopDiscardTrueShiftsElements
VAR
	discardBuffer : DINT;
END_VAR
IF TestSuite.Test(__POUNAME()).ExecuteTest() THEN
	// Arrange
	fbAnyBuffer.Clear();
	RawBuffer[TEST_LL+0] := 10;
	RawBuffer[TEST_LL+1] := 20;
	RawBuffer[TEST_LL+2] := 30;
	RawBuffer[TEST_LL+3] := 40;
	fbAnyBuffer.Metadata.elementCount := 4;

	// Act - Pop with discard=TRUE
	Success := fbAnyBuffer.PopLeft(element := discardBuffer, popDiscard := TRUE);

	// Assert - Elements shifted left correctly
	TestSuite.Test(__POUNAME()).AssertEqual(TEST_BOOL_TRUE, Success);
	TEST_DINT := 20;
	TestSuite.Test(__POUNAME()).AssertEqual(TEST_DINT, RawBuffer[TEST_LL+0]);
	TEST_DINT := 30;
	TestSuite.Test(__POUNAME()).AssertEqual(TEST_DINT, RawBuffer[TEST_LL+1]);
	TEST_DINT := 40;
	TestSuite.Test(__POUNAME()).AssertEqual(TEST_DINT, RawBuffer[TEST_LL+2]);
	TEST_DINT := 0;  // Last element cleared
	TestSuite.Test(__POUNAME()).AssertEqual(TEST_DINT, RawBuffer[TEST_LL+3]);
END_IF
END_METHOD

// No error when element size is wrong and popDiscard=TRUE
METHOD PopDiscardTrueSkipsTypeCheck
VAR
	wrongSizeBuffer : BYTE;  // Only 1 byte, but buffer expects DINT (4 bytes)
END_VAR
IF TestSuite.Test(__POUNAME()).ExecuteTest() THEN
	// Arrange
	fbAnyBuffer.Clear();
	RawBuffer[TEST_LL+0] := 100;
	RawBuffer[TEST_LL+1] := 200;
	fbAnyBuffer.Metadata.elementCount := 2;
	wrongSizeBuffer := 0;

	// Act - Pop with wrong type but popDiscard=TRUE (should succeed)
	Success := fbAnyBuffer.PopLeft(element := wrongSizeBuffer, popDiscard := TRUE);

	// Assert - Should succeed despite type mismatch
	TestSuite.Test(__POUNAME()).AssertEqual(TEST_BOOL_TRUE, Success);
	TEST_DINT := 1;
	TestSuite.Test(__POUNAME()).AssertEqual(TEST_DINT, fbAnyBuffer.Metadata.elementCount);
END_IF
END_METHOD

// PopLeft with wrong type succeeds when popDiscard=TRUE
METHOD PopDiscardWithWrongTypeSucceeds
VAR
	wrongTypeBuffer : INT;  // 2 bytes instead of 4
END_VAR
IF TestSuite.Test(__POUNAME()).ExecuteTest() THEN
	// Arrange
	fbAnyBuffer.Clear();
	RawBuffer[TEST_LL+0] := 999;
	RawBuffer[TEST_LL+1] := 888;
	fbAnyBuffer.Metadata.elementCount := 2;
	wrongTypeBuffer := 0;

	// Act - Pop with wrong type but popDiscard=TRUE
	Success := fbAnyBuffer.PopLeft(element := wrongTypeBuffer, popDiscard := TRUE);

	// Assert - Should succeed
	TestSuite.Test(__POUNAME()).AssertEqual(TEST_BOOL_TRUE, Success);
	TEST_DINT := 1;
	TestSuite.Test(__POUNAME()).AssertEqual(TEST_DINT, fbAnyBuffer.Metadata.elementCount);
	// Buffer shifted correctly
	TEST_DINT := 888;
	TestSuite.Test(__POUNAME()).AssertEqual(TEST_DINT, RawBuffer[TEST_LL+0]);
END_IF
END_METHOD

// PopLeft on empty buffer returns FALSE and does not modify buffer
METHOD PopFromEmptyBuffer
IF TestSuite.Test(__POUNAME()).ExecuteTest() THEN
	// Arrange - Clear buffer (elementCount = 0)
	fbAnyBuffer.Clear();
	ReturnedElement := 999;  // Set to non-zero to verify it is NOT overwritten

	// Act - Pop from empty buffer
	Success := fbAnyBuffer.PopLeft(element := ReturnedElement);

	// Assert - Should fail because buffer is empty
	TestSuite.Test(__POUNAME()).AssertEqual(TEST_BOOL_FALSE, Success);

	// Element should remain unchanged (999) since pop failed
	TEST_DINT := 999;
	TestSuite.Test(__POUNAME()).AssertEqual(TEST_DINT, ReturnedElement);

	// All buffer positions should remain 0
	TEST_DINT := 0;
	TestSuite.Test(__POUNAME()).AssertEqual(TEST_DINT, RawBuffer[TEST_LL+0]);
	TestSuite.Test(__POUNAME()).AssertEqual(TEST_DINT, RawBuffer[TEST_LL+1]);
	TestSuite.Test(__POUNAME()).AssertEqual(TEST_DINT, RawBuffer[TEST_LL+2]);
	TestSuite.Test(__POUNAME()).AssertEqual(TEST_DINT, RawBuffer[TEST_LL+3]);
	TestSuite.Test(__POUNAME()).AssertEqual(TEST_DINT, RawBuffer[TEST_LL+4]);
END_IF
END_METHOD

// PopLeft when buffer contains exactly one element
METHOD PopSingleElement
IF TestSuite.Test(__POUNAME()).ExecuteTest() THEN
	// Arrange - Only first element has data
	fbAnyBuffer.Clear();
	RawBuffer[TEST_LL+0] := 42;
	fbAnyBuffer.Metadata.elementCount := 1;
	ReturnedElement := 0;

	// Act
	Success := fbAnyBuffer.PopLeft(element := ReturnedElement);

	// Assert - Should retrieve the single element
	TestSuite.Test(__POUNAME()).AssertEqual(TEST_BOOL_TRUE, Success);
	TEST_DINT := 42;
	TestSuite.Test(__POUNAME()).AssertEqual(TEST_DINT, ReturnedElement);

	// Buffer should now be completely empty
	TEST_DINT := 0;
	TestSuite.Test(__POUNAME()).AssertEqual(TEST_DINT, RawBuffer[TEST_LL+0]);
	TestSuite.Test(__POUNAME()).AssertEqual(TEST_DINT, RawBuffer[TEST_LL+1]);
	TestSuite.Test(__POUNAME()).AssertEqual(TEST_DINT, RawBuffer[TEST_LL+2]);
	TestSuite.Test(__POUNAME()).AssertEqual(TEST_DINT, RawBuffer[TEST_LL+3]);
	TestSuite.Test(__POUNAME()).AssertEqual(TEST_DINT, RawBuffer[TEST_LL+4]);
END_IF
END_METHOD

// PopLeft can pop all elements until buffer is empty
METHOD PopUntilEmpty
VAR
	i : INT;
	ReturnedElement : DINT;
END_VAR
IF TestSuite.Test(__POUNAME()).ExecuteTest() THEN
	// Arrange - Fill buffer completely
	fbAnyBuffer.Clear();
	FOR i := 1 TO 5 DO
		AppendedElement := TO_DINT(i * 100);
		fbAnyBuffer.PushRight(element := AppendedElement);
	END_FOR

	// Act - Pop all elements
	FOR i := 1 TO 5 DO
		Success := fbAnyBuffer.PopLeft(element := ReturnedElement);
		TestSuite.Test(__POUNAME()).AssertEqual(TEST_BOOL_TRUE, Success);
		TEST_DINT := TO_DINT(i * 100);
		TestSuite.Test(__POUNAME()).AssertEqual(TEST_DINT, ReturnedElement);
	END_FOR

	// Assert - Buffer should be empty
	TEST_DINT := 0;
	TestSuite.Test(__POUNAME()).AssertEqual(TEST_DINT, fbAnyBuffer.Metadata.elementCount);
END_IF
END_METHOD

// PopLeft retrieves the first element from the buffer
METHOD RetrievesFirstElement
IF TestSuite.Test(__POUNAME()).ExecuteTest() THEN
	// Arrange
	fbAnyBuffer.Clear();
	RawBuffer[TEST_LL+0] := 100;
	RawBuffer[TEST_LL+1] := 200;
	RawBuffer[TEST_LL+2] := 300;
	RawBuffer[TEST_LL+3] := 400;
	RawBuffer[TEST_LL+4] := 500;
	fbAnyBuffer.Metadata.elementCount := 5;
	ReturnedElement := 0;

	// Act
	Success := fbAnyBuffer.PopLeft(element := ReturnedElement);

	// Assert
	TestSuite.Test(__POUNAME()).AssertEqual(TEST_BOOL_TRUE, Success);
	TEST_DINT := 100;
	TestSuite.Test(__POUNAME()).AssertEqual(TEST_DINT, ReturnedElement);
END_IF
END_METHOD

// Method returns TRUE when pop succeeds
METHOD ReturnsTrueOnSuccess
IF TestSuite.Test(__POUNAME()).ExecuteTest() THEN
	// Arrange
	fbAnyBuffer.Clear();
	RawBuffer[TEST_LL+0] := 100;
	RawBuffer[TEST_LL+1] := 200;
	fbAnyBuffer.Metadata.elementCount := 2;

	// Act
	Success := fbAnyBuffer.PopLeft(element := ReturnedElement);

	// Assert
	TestSuite.Test(__POUNAME()).AssertEqual(TEST_BOOL_TRUE, Success);
END_IF
END_METHOD

// PopLeft shifts all elements one position to the left
METHOD ShiftsElements
IF TestSuite.Test(__POUNAME()).ExecuteTest() THEN
	// Arrange
	fbAnyBuffer.Clear();
	RawBuffer[TEST_LL+0] := 100;
	RawBuffer[TEST_LL+1] := 200;
	RawBuffer[TEST_LL+2] := 300;
	RawBuffer[TEST_LL+3] := 400;
	RawBuffer[TEST_LL+4] := 500;
	fbAnyBuffer.Metadata.elementCount := 5;
	ReturnedElement := 0;

	// Act
	Success := fbAnyBuffer.PopLeft(element := ReturnedElement);

	// Assert - Elements should be shifted left
	TEST_DINT := 200;
	TestSuite.Test(__POUNAME()).AssertEqual(TEST_DINT, RawBuffer[TEST_LL+0]);
	TEST_DINT := 300;
	TestSuite.Test(__POUNAME()).AssertEqual(TEST_DINT, RawBuffer[TEST_LL+1]);
	TEST_DINT := 400;
	TestSuite.Test(__POUNAME()).AssertEqual(TEST_DINT, RawBuffer[TEST_LL+2]);
	TEST_DINT := 500;
	TestSuite.Test(__POUNAME()).AssertEqual(TEST_DINT, RawBuffer[TEST_LL+3]);
END_IF
END_METHOD

// PopLeft returns FALSE when element size doesn't match buffer element size
METHOD WrongSize
IF TestSuite.Test(__POUNAME()).ExecuteTest() THEN
	// Arrange
	fbAnyBuffer.Clear();
	RawBuffer[TEST_LL+0] := 100;
	fbAnyBuffer.Metadata.elementCount := 1;
	WrongSizeElement := 0;

	// Act - Pass an INT (2 bytes) to a DINT buffer (4 bytes)
	Success := fbAnyBuffer.PopLeft(element := WrongSizeElement);

	// Assert
	TestSuite.Test(__POUNAME()).AssertEqual(TEST_BOOL_FALSE, Success);
END_IF
END_METHOD

END_PROGRAM

// ---- UnitTests/AnyBuffer/TEST_AnyBuffer_PopRight.TcPOU
PROGRAM TEST_AnyBuffer_PopRight
VAR
	// Loop counter
	i						: DINT;
END_VAR

RetrievesLastElement();
DoesNotShiftElements();
ClearsLastElement();
DecrementsElementCount();
ReturnsTrueOnSuccess();
WrongSize();
EmptyElement();
PopFromEmptyBuffer();
PopSingleElement();
ConsecutivePops();
PopAfterAppendRight();
PopAfterAppendLeft();
PopUntilEmpty();
ElementOrderPreserved();
PopDiscardTrue();
PopDiscardTrueSkipsTypeCheck();
PopDiscardTrueNoShift();
PopDiscardTrueDecrementsCount();
PopDiscardFalseRetrievesValue();
PopDiscardFalseValidatesType();
PopDiscardWithWrongTypeSucceeds();
PopDiscardReturnsTrueOnSuccess();

// PopRight clears the last element of the buffer
METHOD ClearsLastElement
IF TestSuite.Test(__POUNAME()).ExecuteTest() THEN
	// Arrange
	fbAnyBuffer.Clear();
	RawBuffer[TEST_LL+0] := 100;
	RawBuffer[TEST_LL+1] := 200;
	RawBuffer[TEST_LL+2] := 300;
	RawBuffer[TEST_LL+3] := 400;
	RawBuffer[TEST_LL+4] := 500;
	fbAnyBuffer.Metadata.elementCount := 5;
	ReturnedElement := 0;

	// Act
	Success := fbAnyBuffer.PopRight(element := ReturnedElement);

	// Assert - Last element should be cleared (0)
	TEST_DINT := 0;
	TestSuite.Test(__POUNAME()).AssertEqual(TEST_DINT, RawBuffer[TEST_LL+4]);
END_IF
END_METHOD

// PopRight multiple times maintains correct order (LIFO)
METHOD ConsecutivePops
VAR
	pop1 : DINT;
	pop2 : DINT;
	pop3 : DINT;
END_VAR
IF TestSuite.Test(__POUNAME()).ExecuteTest() THEN
	// Arrange - Fill buffer with sequential values
	fbAnyBuffer.Clear();
	RawBuffer[TEST_LL+0] := 10;
	RawBuffer[TEST_LL+1] := 20;
	RawBuffer[TEST_LL+2] := 30;
	RawBuffer[TEST_LL+3] := 40;
	RawBuffer[TEST_LL+4] := 50;
	fbAnyBuffer.Metadata.elementCount := 5;

	// Act - Pop three times consecutively from right
	fbAnyBuffer.PopRight(element := pop1);
	fbAnyBuffer.PopRight(element := pop2);
	fbAnyBuffer.PopRight(element := pop3);

	// Assert - Elements should be retrieved in reverse order (LIFO)
	TEST_DINT := 50;
	TestSuite.Test(__POUNAME()).AssertEqual(TEST_DINT, pop1);
	TEST_DINT := 40;
	TestSuite.Test(__POUNAME()).AssertEqual(TEST_DINT, pop2);
	TEST_DINT := 30;
	TestSuite.Test(__POUNAME()).AssertEqual(TEST_DINT, pop3);

	// Remaining buffer state: [10, 20, 0, 0, 0]
	TEST_DINT := 10;
	TestSuite.Test(__POUNAME()).AssertEqual(TEST_DINT, RawBuffer[TEST_LL+0]);
	TEST_DINT := 20;
	TestSuite.Test(__POUNAME()).AssertEqual(TEST_DINT, RawBuffer[TEST_LL+1]);
	TEST_DINT := 0;
	TestSuite.Test(__POUNAME()).AssertEqual(TEST_DINT, RawBuffer[TEST_LL+2]);
	TestSuite.Test(__POUNAME()).AssertEqual(TEST_DINT, RawBuffer[TEST_LL+3]);
	TestSuite.Test(__POUNAME()).AssertEqual(TEST_DINT, RawBuffer[TEST_LL+4]);
	TEST_DINT := 2;
	TestSuite.Test(__POUNAME()).AssertEqual(TEST_DINT, fbAnyBuffer.Metadata.elementCount);
END_IF
END_METHOD

// PopRight decreases elementCount by 1
METHOD DecrementsElementCount
IF TestSuite.Test(__POUNAME()).ExecuteTest() THEN
	// Arrange
	fbAnyBuffer.Clear();
	RawBuffer[TEST_LL+0] := 100;
	RawBuffer[TEST_LL+1] := 200;
	RawBuffer[TEST_LL+2] := 300;
	fbAnyBuffer.Metadata.elementCount := 3;

	// Act
	Success := fbAnyBuffer.PopRight(element := ReturnedElement);

	// Assert - elementCount should be decremented from 3 to 2
	TEST_DINT := 2;
	TestSuite.Test(__POUNAME()).AssertEqual(TEST_DINT, fbAnyBuffer.Metadata.elementCount);
END_IF
END_METHOD

// PopRight does not shift any remaining elements
METHOD DoesNotShiftElements
IF TestSuite.Test(__POUNAME()).ExecuteTest() THEN
	// Arrange
	fbAnyBuffer.Clear();
	RawBuffer[TEST_LL+0] := 100;
	RawBuffer[TEST_LL+1] := 200;
	RawBuffer[TEST_LL+2] := 300;
	RawBuffer[TEST_LL+3] := 400;
	RawBuffer[TEST_LL+4] := 500;
	fbAnyBuffer.Metadata.elementCount := 5;
	ReturnedElement := 0;

	// Act
	Success := fbAnyBuffer.PopRight(element := ReturnedElement);

	// Assert - Elements should remain at their original positions
	TEST_DINT := 100;
	TestSuite.Test(__POUNAME()).AssertEqual(TEST_DINT, RawBuffer[TEST_LL+0]);
	TEST_DINT := 200;
	TestSuite.Test(__POUNAME()).AssertEqual(TEST_DINT, RawBuffer[TEST_LL+1]);
	TEST_DINT := 300;
	TestSuite.Test(__POUNAME()).AssertEqual(TEST_DINT, RawBuffer[TEST_LL+2]);
	TEST_DINT := 400;
	TestSuite.Test(__POUNAME()).AssertEqual(TEST_DINT, RawBuffer[TEST_LL+3]);
END_IF
END_METHOD

// PopRight preserves remaining element positions
METHOD ElementOrderPreserved
IF TestSuite.Test(__POUNAME()).ExecuteTest() THEN
	// Arrange
	fbAnyBuffer.Clear();
	RawBuffer[TEST_LL+0] := 111;
	RawBuffer[TEST_LL+1] := 222;
	RawBuffer[TEST_LL+2] := 333;
	RawBuffer[TEST_LL+3] := 444;
	RawBuffer[TEST_LL+4] := 555;
	fbAnyBuffer.Metadata.elementCount := 5;

	// Act - Pop last two elements
	fbAnyBuffer.PopRight(element := ReturnedElement);
	fbAnyBuffer.PopRight(element := ReturnedElement);

	// Assert - First three elements should remain at original positions
	TEST_DINT := 111;
	TestSuite.Test(__POUNAME()).AssertEqual(TEST_DINT, RawBuffer[TEST_LL+0]);
	TEST_DINT := 222;
	TestSuite.Test(__POUNAME()).AssertEqual(TEST_DINT, RawBuffer[TEST_LL+1]);
	TEST_DINT := 333;
	TestSuite.Test(__POUNAME()).AssertEqual(TEST_DINT, RawBuffer[TEST_LL+2]);

	// Last two positions should be cleared
	TEST_DINT := 0;
	TestSuite.Test(__POUNAME()).AssertEqual(TEST_DINT, RawBuffer[TEST_LL+3]);
	TestSuite.Test(__POUNAME()).AssertEqual(TEST_DINT, RawBuffer[TEST_LL+4]);

	TEST_DINT := 3;
	TestSuite.Test(__POUNAME()).AssertEqual(TEST_DINT, fbAnyBuffer.Metadata.elementCount);
END_IF
END_METHOD

// PopRight with zero-sized element just clears without copying
METHOD EmptyElement
VAR
	EmptyAny				: __SYSTEM.AnyType;
END_VAR
IF TestSuite.Test(__POUNAME()).ExecuteTest() THEN
	// Arrange
	fbAnyBuffer.Clear();
	RawBuffer[TEST_LL+0] := 100;
	RawBuffer[TEST_LL+1] := 200;
	RawBuffer[TEST_LL+2] := 300;
	fbAnyBuffer.Metadata.elementCount := 3;
	fbAnyBuffer.Metadata.capacity := 2;

	// Initialize empty AnyType (size = 0)
	EmptyAny.pValue := 0;
	EmptyAny.diSize := 0;

	// Act - Call with zero-sized element
	Success := fbAnyBuffer.PopRight(element := EmptyAny);

	// Assert - Should NOT succeed and clear last element
	TestSuite.Test(__POUNAME()).AssertEqual(TEST_BOOL_FALSE, Success);
	TEST_DINT := 3;
	TestSuite.Test(__POUNAME()).AssertEqual(TEST_DINT, fbAnyBuffer.Metadata.elementCount);
	TEST_DINT := 300;
	TestSuite.Test(__POUNAME()).AssertEqual(TEST_DINT, RawBuffer[TEST_LL+2]);
END_IF
END_METHOD

// PopRight with AppendLeft demonstrates FIFO behavior
METHOD PopAfterAppendLeft
VAR
	ReturnedElement : DINT;
	testElement : DINT;
END_VAR
IF TestSuite.Test(__POUNAME()).ExecuteTest() THEN
	// Arrange
	fbAnyBuffer.Clear();

	// Act - Append left and Pop right (FIFO: First In First Out)
	testElement := DINT#100;
	fbAnyBuffer.PushLeft(element := testElement);  // [100]
	testElement := DINT#200;
	fbAnyBuffer.PushLeft(element := testElement);  // [200, 100]
	testElement := DINT#300;
	fbAnyBuffer.PushLeft(element := testElement);  // [300, 200, 100]
	fbAnyBuffer.PopRight(element := ReturnedElement); // Pop 100 (first appended)

	// Assert - Should pop the first appended value (100)
	TEST_DINT := 100;
	TestSuite.Test(__POUNAME()).AssertEqual(TEST_DINT, ReturnedElement);

	// Buffer should now be [300, 200]
	TEST_DINT := 300;
	TestSuite.Test(__POUNAME()).AssertEqual(TEST_DINT, RawBuffer[TEST_LL+0]);
	TEST_DINT := 200;
	TestSuite.Test(__POUNAME()).AssertEqual(TEST_DINT, RawBuffer[TEST_LL+1]);
	TEST_DINT := 2;
	TestSuite.Test(__POUNAME()).AssertEqual(TEST_DINT, fbAnyBuffer.Metadata.elementCount);
END_IF
END_METHOD

// PopRight with AppendRight demonstrates LIFO behavior
METHOD PopAfterAppendRight
VAR
	ReturnedElement : DINT;
	testElement : DINT;
END_VAR
IF TestSuite.Test(__POUNAME()).ExecuteTest() THEN
	// Arrange
	fbAnyBuffer.Clear();

	// Act - Append and Pop from right (LIFO: Last In First Out)
	testElement := DINT#100;
	fbAnyBuffer.PushRight(element := testElement);  // [100]
	testElement := DINT#200;
	fbAnyBuffer.PushRight(element := testElement);  // [100, 200]
	testElement := DINT#300;
	fbAnyBuffer.PushRight(element := testElement);  // [100, 200, 300]
	fbAnyBuffer.PopRight(element := ReturnedElement);  // Pop 300

	// Assert - Should pop the last appended value (300)
	TEST_DINT := 300;
	TestSuite.Test(__POUNAME()).AssertEqual(TEST_DINT, ReturnedElement);

	// Buffer should now be [100, 200]
	TEST_DINT := 100;
	TestSuite.Test(__POUNAME()).AssertEqual(TEST_DINT, RawBuffer[TEST_LL+0]);
	TEST_DINT := 200;
	TestSuite.Test(__POUNAME()).AssertEqual(TEST_DINT, RawBuffer[TEST_LL+1]);
	TEST_DINT := 2;
	TestSuite.Test(__POUNAME()).AssertEqual(TEST_DINT, fbAnyBuffer.Metadata.elementCount);
END_IF
END_METHOD

// Element value is copied when popDiscard=FALSE (default)
METHOD PopDiscardFalseRetrievesValue
IF TestSuite.Test(__POUNAME()).ExecuteTest() THEN
	// Arrange
	fbAnyBuffer.Clear();
	RawBuffer[TEST_LL+0] := 123;
	RawBuffer[TEST_LL+1] := 456;
	fbAnyBuffer.Metadata.elementCount := 2;
	ReturnedElement := 0;

	// Act - Pop with explicit popDiscard=FALSE
	Success := fbAnyBuffer.PopRight(element := ReturnedElement, popDiscard := FALSE);

	// Assert - Value is retrieved (last element)
	TestSuite.Test(__POUNAME()).AssertEqual(TEST_BOOL_TRUE, Success);
	TEST_DINT := 456;
	TestSuite.Test(__POUNAME()).AssertEqual(TEST_DINT, ReturnedElement);
END_IF
END_METHOD

// Type checking occurs when popDiscard=FALSE
METHOD PopDiscardFalseValidatesType
IF TestSuite.Test(__POUNAME()).ExecuteTest() THEN
	// Arrange
	fbAnyBuffer.Clear();
	RawBuffer[TEST_LL+0] := 100;
	fbAnyBuffer.Metadata.elementCount := 1;
	WrongSizeElement := 0;

	// Act - Pop with wrong type and popDiscard=FALSE (should fail)
	Success := fbAnyBuffer.PopRight(element := WrongSizeElement, popDiscard := FALSE);

	// Assert - Should fail due to type mismatch
	TestSuite.Test(__POUNAME()).AssertEqual(TEST_BOOL_FALSE, Success);
	// Element count should remain unchanged (pop failed)
	TEST_DINT := 1;
	TestSuite.Test(__POUNAME()).AssertEqual(TEST_DINT, fbAnyBuffer.Metadata.elementCount);
END_IF
END_METHOD

// Method returns TRUE when popDiscard=TRUE succeeds
METHOD PopDiscardReturnsTrueOnSuccess
VAR
	discardBuffer : DINT;
END_VAR
IF TestSuite.Test(__POUNAME()).ExecuteTest() THEN
	// Arrange
	fbAnyBuffer.Clear();
	RawBuffer[TEST_LL+0] := 777;
	fbAnyBuffer.Metadata.elementCount := 1;

	// Act
	Success := fbAnyBuffer.PopRight(element := discardBuffer, popDiscard := TRUE);

